  PROC DrawPart142()
    MoveL Offs(pOrigin,284.64,277.94,6.00),vTravel,z5,tPen\WObj:=wPaper;
    MoveL Offs(pOrigin,284.64,277.94,0.00),v60,z0,tPen\WObj:=wPaper;
    MoveL Offs(pOrigin,280.81,277.94,0.00),v40,fine,tPen\WObj:=wPaper;
    MoveL Offs(pOrigin,280.81,277.94,6.00),v60,z5,tPen\WObj:=wPaper;
    MoveL Offs(pOrigin,279.25,279.53,6.00),vTravel,z5,tPen\WObj:=wPaper;
    MoveL Offs(pOrigin,279.25,279.53,0.00),v60,z0,tPen\WObj:=wPaper;
    MoveL Offs(pOrigin,292.32,266.46,0.00),v40,z0,tPen\WObj:=wPaper;
    MoveL Offs(pOrigin,292.92,267.36,0.00),v40,z0,tPen\WObj:=wPaper;
    MoveL Offs(pOrigin,278.80,281.48,0.00),v40,z0,tPen\WObj:=wPaper;
    MoveL Offs(pOrigin,279.75,281.54,0.00),v40,z0,tPen\WObj:=wPaper;
    MoveL Offs(pOrigin,297.48,299.27,0.00),v40,z0,tPen\WObj:=wPaper;
    MoveL Offs(pOrigin,296.96,299.06,0.00),v40,z0,tPen\WObj:=wPaper;
    MoveL Offs(pOrigin,291.23,299.06,0.00),v40,z0,tPen\WObj:=wPaper;
    MoveL Offs(pOrigin,291.23,298.04,0.00),v40,z0,tPen\WObj:=wPaper;
    MoveL Offs(pOrigin,293.99,297.61,0.00),v40,z0,tPen\WObj:=wPaper;
    MoveL Offs(pOrigin,293.99,297.61,0.00),v40,z0,tPen\WObj:=wPaper;
    MoveL Offs(pOrigin,293.56,296.83,0.00),v40,z0,tPen\WObj:=wPaper;
    MoveL Offs(pOrigin,292.08,296.76,0.00),v40,z0,tPen\WObj:=wPaper;
    MoveL Offs(pOrigin,291.23,297.61,0.00),v40,fine,tPen\WObj:=wPaper;
    MoveL Offs(pOrigin,291.23,297.61,6.00),v60,z5,tPen\WObj:=wPaper;
    MoveL Offs(pOrigin,292.92,298.01,6.00),vTravel,z5,tPen\WObj:=wPaper;
    MoveL Offs(pOrigin,292.92,298.01,0.00),v60,z0,tPen\WObj:=wPaper;
    MoveL Offs(pOrigin,296.96,298.01,0.00),v40,z0,tPen\WObj:=wPaper;
    MoveL Offs(pOrigin,297.48,297.77,0.00),v40,z0,tPen\WObj:=wPaper;
    MoveL Offs(pOrigin,279.90,280.19,0.00),v40,fine,tPen\WObj:=wPaper;
    MoveL Offs(pOrigin,279.90,280.19,6.00),v60,z5,tPen\WObj:=wPaper;
    MoveL Offs(pOrigin,281.97,281.89,6.00),vTravel,z5,tPen\WObj:=wPaper;
    MoveL Offs(pOrigin,281.97,281.89,0.00),v60,z0,tPen\WObj:=wPaper;
    MoveL Offs(pOrigin,281.97,275.72,0.00),v40,z0,tPen\WObj:=wPaper;
    MoveL Offs(pOrigin,281.66,275.83,0.00),v40,z0,tPen\WObj:=wPaper;
    MoveL Offs(pOrigin,299.51,275.83,0.00),v40,z0,tPen\WObj:=wPaper;
    MoveL Offs(pOrigin,299.96,276.36,0.00),v40,z0,tPen\WObj:=wPaper;
    MoveL Offs(pOrigin,297.40,273.80,0.00),v40,z0,tPen\WObj:=wPaper;
    MoveL Offs(pOrigin,297.81,274.66,0.00),v40,z0,tPen\WObj:=wPaper;
    MoveL Offs(pOrigin,297.81,280.19,0.00),v40,z0,tPen\WObj:=wPaper;
    MoveL Offs(pOrigin,298.45,280.06,0.00),v40,z0,tPen\WObj:=wPaper;
    MoveL Offs(pOrigin,285.06,280.06,0.00),v40,z0,tPen\WObj:=wPaper;
    MoveL Offs(pOrigin,285.27,279.76,0.00),v40,z0,tPen\WObj:=wPaper;
    MoveL Offs(pOrigin,284.85,280.19,0.00),v40,z0,tPen\WObj:=wPaper;
    MoveL Offs(pOrigin,285.27,279.76,0.00),v40,z0,tPen\WObj:=wPaper;
    MoveL Offs(pOrigin,285.13,280.61,0.00),v40,z0,tPen\WObj:=wPaper;
    MoveL Offs(pOrigin,285.13,282.10,0.00),v40,z0,tPen\WObj:=wPaper;
    MoveL Offs(pOrigin,285.06,283.22,0.00),v40,z0,tPen\WObj:=wPaper;
    MoveL Offs(pOrigin,280.60,283.22,0.00),v40,z0,tPen\WObj:=wPaper;
    MoveL Offs(pOrigin,280.60,284.28,0.00),v40,z0,tPen\WObj:=wPaper;
    MoveL Offs(pOrigin,284.85,284.28,0.00),v40,z0,tPen\WObj:=wPaper;
    MoveL Offs(pOrigin,284.85,284.65,0.00),v40,z0,tPen\WObj:=wPaper;
    MoveL Offs(pOrigin,283.72,286.99,0.00),v40,z0,tPen\WObj:=wPaper;
    MoveL Offs(pOrigin,285.70,287.20,0.00),v40,z0,tPen\WObj:=wPaper;
    MoveL Offs(pOrigin,285.27,287.45,0.00),v40,z0,tPen\WObj:=wPaper;
    MoveL Offs(pOrigin,280.81,287.45,0.00),v40,z0,tPen\WObj:=wPaper;
    MoveL Offs(pOrigin,280.60,288.50,0.00),v40,z0,tPen\WObj:=wPaper;
    MoveL Offs(pOrigin,284.21,288.50,0.00),v40,z0,tPen\WObj:=wPaper;
    MoveL Offs(pOrigin,284.85,288.26,0.00),v40,z0,tPen\WObj:=wPaper;
    MoveL Offs(pOrigin,284.42,288.69,0.00),v40,z0,tPen\WObj:=wPaper;
    MoveL Offs(pOrigin,284.85,288.26,0.00),v40,fine,tPen\WObj:=wPaper;
    MoveL Offs(pOrigin,284.85,288.26,6.00),v60,z5,tPen\WObj:=wPaper;
    MoveL Offs(pOrigin,285.13,286.99,6.00),vTravel,z5,tPen\WObj:=wPaper;
    MoveL Offs(pOrigin,285.13,286.99,0.00),v60,z0,tPen\WObj:=wPaper;
    MoveL Offs(pOrigin,285.13,285.92,0.00),v40,z0,tPen\WObj:=wPaper;
    MoveL Offs(pOrigin,286.19,285.50,0.00),v40,z0,tPen\WObj:=wPaper;
    MoveL Offs(pOrigin,286.19,286.56,0.00),v40,fine,tPen\WObj:=wPaper;
    MoveL Offs(pOrigin,286.19,286.56,6.00),v60,z5,tPen\WObj:=wPaper;
    MoveL Offs(pOrigin,287.61,286.39,6.00),vTravel,z5,tPen\WObj:=wPaper;
    MoveL Offs(pOrigin,287.61,286.39,0.00),v60,z0,tPen\WObj:=wPaper;
    MoveL Offs(pOrigin,281.02,286.39,0.00),v40,z0,tPen\WObj:=wPaper;
    MoveL Offs(pOrigin,280.81,285.34,0.00),v40,z0,tPen\WObj:=wPaper;
    MoveL Offs(pOrigin,289.10,285.34,0.00),v40,z0,tPen\WObj:=wPaper;
    MoveL Offs(pOrigin,288.67,286.14,0.00),v40,z0,tPen\WObj:=wPaper;
    MoveL Offs(pOrigin,289.10,286.56,0.00),v40,z0,tPen\WObj:=wPaper;
    MoveL Offs(pOrigin,289.74,286.56,0.00),v40,z0,tPen\WObj:=wPaper;
    MoveL Offs(pOrigin,289.95,286.99,0.00),v40,z0,tPen\WObj:=wPaper;
    MoveL Offs(pOrigin,289.95,286.99,0.00),v40,z0,tPen\WObj:=wPaper;
    MoveL Offs(pOrigin,286.98,288.48,0.00),v40,z0,tPen\WObj:=wPaper;
    MoveL Offs(pOrigin,287.40,288.50,0.00),v40,z0,tPen\WObj:=wPaper;
    MoveL Offs(pOrigin,289.95,288.50,0.00),v40,z0,tPen\WObj:=wPaper;
    MoveL Offs(pOrigin,290.16,289.11,0.00),v40,z0,tPen\WObj:=wPaper;
    MoveL Offs(pOrigin,293.99,289.96,0.00),v40,z0,tPen\WObj:=wPaper;
    MoveL Offs(pOrigin,294.20,289.56,0.00),v40,z0,tPen\WObj:=wPaper;
    MoveL Offs(pOrigin,298.02,289.56,0.00),v40,fine,tPen\WObj:=wPaper;
    MoveL Offs(pOrigin,298.02,289.56,6.00),v60,z5,tPen\WObj:=wPaper;
    MoveL Offs(pOrigin,299.00,288.16,6.00),vTravel,z5,tPen\WObj:=wPaper;
    MoveL Offs(pOrigin,299.00,288.16,0.00),v60,z0,tPen\WObj:=wPaper;
    MoveL Offs(pOrigin,261.88,325.27,0.00),v40,z0,tPen\WObj:=wPaper;
    MoveL Offs(pOrigin,261.14,324.53,0.00),v40,z0,tPen\WObj:=wPaper;
    MoveL Offs(pOrigin,299.00,286.66,0.00),v40,z0,tPen\WObj:=wPaper;
    MoveL Offs(pOrigin,298.49,286.84,0.00),v40,z0,tPen\WObj:=wPaper;
    MoveL Offs(pOrigin,282.26,270.61,0.00),v40,z0,tPen\WObj:=wPaper;
    MoveL Offs(pOrigin,282.51,271.26,0.00),v40,z0,tPen\WObj:=wPaper;
    MoveL Offs(pOrigin,284.00,269.49,0.00),v40,z0,tPen\WObj:=wPaper;
    MoveL Offs(pOrigin,285.70,269.99,0.00),v40,z0,tPen\WObj:=wPaper;
    MoveL Offs(pOrigin,286.55,269.14,0.00),v40,z0,tPen\WObj:=wPaper;
    MoveL Offs(pOrigin,286.98,266.38,0.00),v40,z0,tPen\WObj:=wPaper;
    MoveL Offs(pOrigin,286.76,265.31,0.00),v40,z0,tPen\WObj:=wPaper;
    MoveL Offs(pOrigin,287.40,264.25,0.00),v40,fine,tPen\WObj:=wPaper;
    MoveL Offs(pOrigin,287.40,264.25,6.00),v60,z5,tPen\WObj:=wPaper;
    MoveL Offs(pOrigin,291.29,263.02,6.00),vTravel,z5,tPen\WObj:=wPaper;
    MoveL Offs(pOrigin,291.29,263.02,0.00),v60,z0,tPen\WObj:=wPaper;
    MoveL Offs(pOrigin,280.32,273.99,0.00),v40,z0,tPen\WObj:=wPaper;
    MoveL Offs(pOrigin,280.76,275.03,0.00),v40,z0,tPen\WObj:=wPaper;
    MoveL Offs(pOrigin,291.58,264.21,0.00),v40,fine,tPen\WObj:=wPaper;
    MoveL Offs(pOrigin,291.58,264.21,6.00),v60,z5,tPen\WObj:=wPaper;
    MoveL Offs(pOrigin,290.92,261.35,6.00),vTravel,z5,tPen\WObj:=wPaper;
    MoveL Offs(pOrigin,290.92,261.35,0.00),v60,z0,tPen\WObj:=wPaper;
    MoveL Offs(pOrigin,288.37,258.79,0.00),v40,fine,tPen\WObj:=wPaper;
    MoveL Offs(pOrigin,288.37,258.79,6.00),v60,z5,tPen\WObj:=wPaper;
    MoveL Offs(pOrigin,290.02,258.95,6.00),vTravel,z5,tPen\WObj:=wPaper;
    MoveL Offs(pOrigin,290.02,258.95,0.00),v60,z0,tPen\WObj:=wPaper;
    MoveL Offs(pOrigin,291.37,260.30,0.00),v40,z0,tPen\WObj:=wPaper;
    MoveL Offs(pOrigin,292.34,260.47,0.00),v40,z0,tPen\WObj:=wPaper;
    MoveL Offs(pOrigin,278.82,273.99,0.00),v40,fine,tPen\WObj:=wPaper;
    MoveL Offs(pOrigin,278.82,273.99,6.00),v60,z5,tPen\WObj:=wPaper;
    MoveL Offs(pOrigin,277.47,273.85,6.00),vTravel,z5,tPen\WObj:=wPaper;
    MoveL Offs(pOrigin,277.47,273.85,0.00),v60,z0,tPen\WObj:=wPaper;
    MoveL Offs(pOrigin,281.53,269.79,0.00),v40,fine,tPen\WObj:=wPaper;
    MoveL Offs(pOrigin,281.53,269.79,6.00),v60,z5,tPen\WObj:=wPaper;
    MoveL Offs(pOrigin,280.33,269.49,6.00),vTravel,z5,tPen\WObj:=wPaper;
    MoveL Offs(pOrigin,280.33,269.49,0.00),v60,z0,tPen\WObj:=wPaper;
    MoveL Offs(pOrigin,275.97,273.85,0.00),v40,z0,tPen\WObj:=wPaper;
    MoveL Offs(pOrigin,275.92,272.96,0.00),v40,z0,tPen\WObj:=wPaper;
  ENDPROC

  PROC DrawPart143()
    MoveL Offs(pOrigin,274.44,273.39,0.00),v40,fine,tPen\WObj:=wPaper;
    MoveL Offs(pOrigin,274.44,273.39,6.00),v60,z5,tPen\WObj:=wPaper;
    MoveL Offs(pOrigin,273.42,274.91,6.00),vTravel,z5,tPen\WObj:=wPaper;
    MoveL Offs(pOrigin,273.42,274.91,0.00),v60,z0,tPen\WObj:=wPaper;
    MoveL Offs(pOrigin,279.13,269.20,0.00),v40,z0,tPen\WObj:=wPaper;
    MoveL Offs(pOrigin,278.09,268.75,0.00),v40,z0,tPen\WObj:=wPaper;
    MoveL Offs(pOrigin,271.48,275.36,0.00),v40,fine,tPen\WObj:=wPaper;
    MoveL Offs(pOrigin,271.48,275.36,6.00),v60,z5,tPen\WObj:=wPaper;
    MoveL Offs(pOrigin,269.98,275.37,6.00),vTravel,z5,tPen\WObj:=wPaper;
    MoveL Offs(pOrigin,269.98,275.37,0.00),v60,z0,tPen\WObj:=wPaper;
    MoveL Offs(pOrigin,271.93,273.41,0.00),v40,z0,tPen\WObj:=wPaper;
    MoveL Offs(pOrigin,271.48,272.37,0.00),v40,z0,tPen\WObj:=wPaper;
    MoveL Offs(pOrigin,268.03,275.82,0.00),v40,z0,tPen\WObj:=wPaper;
    MoveL Offs(pOrigin,267.30,275.06,0.00),v40,z0,tPen\WObj:=wPaper;
    MoveL Offs(pOrigin,264.89,272.65,0.00),v40,z0,tPen\WObj:=wPaper;
    MoveL Offs(pOrigin,265.51,272.75,0.00),v40,z0,tPen\WObj:=wPaper;
    MoveL Offs(pOrigin,266.58,272.96,0.00),v40,z0,tPen\WObj:=wPaper;
    MoveL Offs(pOrigin,267.00,272.54,0.00),v40,z0,tPen\WObj:=wPaper;
    MoveL Offs(pOrigin,267.00,272.54,0.00),v40,z0,tPen\WObj:=wPaper;
    MoveL Offs(pOrigin,266.79,272.11,0.00),v40,z0,tPen\WObj:=wPaper;
    MoveL Offs(pOrigin,265.73,272.11,0.00),v40,z0,tPen\WObj:=wPaper;
    MoveL Offs(pOrigin,265.51,272.75,0.00),v40,z0,tPen\WObj:=wPaper;
    MoveL Offs(pOrigin,265.51,272.75,0.00),v40,z0,tPen\WObj:=wPaper;
    MoveL Offs(pOrigin,264.02,272.96,0.00),v40,z0,tPen\WObj:=wPaper;
    MoveL Offs(pOrigin,258.92,271.69,0.00),v40,z0,tPen\WObj:=wPaper;
    MoveL Offs(pOrigin,256.38,271.48,0.00),v40,z0,tPen\WObj:=wPaper;
    MoveL Offs(pOrigin,254.68,270.98,0.00),v40,z0,tPen\WObj:=wPaper;
    MoveL Offs(pOrigin,254.18,270.41,0.00),v40,z0,tPen\WObj:=wPaper;
    MoveL Offs(pOrigin,254.68,269.99,0.00),v40,z0,tPen\WObj:=wPaper;
    MoveL Offs(pOrigin,255.95,269.99,0.00),v40,z0,tPen\WObj:=wPaper;
    MoveL Offs(pOrigin,255.95,269.99,0.00),v40,z0,tPen\WObj:=wPaper;
    MoveL Offs(pOrigin,256.16,270.20,0.00),v40,z0,tPen\WObj:=wPaper;
    MoveL Offs(pOrigin,257.01,269.99,0.00),v40,z0,tPen\WObj:=wPaper;
    MoveL Offs(pOrigin,256.65,270.38,0.00),v40,z0,tPen\WObj:=wPaper;
    MoveL Offs(pOrigin,250.34,264.07,0.00),v40,fine,tPen\WObj:=wPaper;
    MoveL Offs(pOrigin,250.34,264.07,6.00),v60,z5,tPen\WObj:=wPaper;
    MoveL Offs(pOrigin,251.53,263.77,6.00),vTravel,z5,tPen\WObj:=wPaper;
    MoveL Offs(pOrigin,251.53,263.77,0.00),v60,z0,tPen\WObj:=wPaper;
    MoveL Offs(pOrigin,257.84,270.08,0.00),v40,z0,tPen\WObj:=wPaper;
    MoveL Offs(pOrigin,257.40,271.13,0.00),v40,z0,tPen\WObj:=wPaper;
    MoveL Offs(pOrigin,262.81,276.54,0.00),v40,z0,tPen\WObj:=wPaper;
    MoveL Offs(pOrigin,262.48,276.89,0.00),v40,z0,tPen\WObj:=wPaper;
    MoveL Offs(pOrigin,268.49,270.88,0.00),v40,z0,tPen\WObj:=wPaper;
    MoveL Offs(pOrigin,268.70,271.05,0.00),v40,z0,tPen\WObj:=wPaper;
    MoveL Offs(pOrigin,269.69,271.33,0.00),v40,z0,tPen\WObj:=wPaper;
    MoveL Offs(pOrigin,270.40,270.84,0.00),v40,z0,tPen\WObj:=wPaper;
    MoveL Offs(pOrigin,270.75,271.05,0.00),v40,z0,tPen\WObj:=wPaper;
    MoveL Offs(pOrigin,270.83,271.69,0.00),v40,z0,tPen\WObj:=wPaper;
    MoveL Offs(pOrigin,271.49,270.87,0.00),v40,z0,tPen\WObj:=wPaper;
    MoveL Offs(pOrigin,266.08,276.28,0.00),v40,z0,tPen\WObj:=wPaper;
    MoveL Offs(pOrigin,265.35,276.10,0.00),v40,z0,tPen\WObj:=wPaper;
    MoveL Offs(pOrigin,261.90,272.64,0.00),v40,z0,tPen\WObj:=wPaper;
    MoveL Offs(pOrigin,261.90,271.50,0.00),v40,z0,tPen\WObj:=wPaper;
    MoveL Offs(pOrigin,257.54,275.85,0.00),v40,z0,tPen\WObj:=wPaper;
    MoveL Offs(pOrigin,257.41,275.63,0.00),v40,z0,tPen\WObj:=wPaper;
    MoveL Offs(pOrigin,252.45,270.67,0.00),v40,fine,tPen\WObj:=wPaper;
    MoveL Offs(pOrigin,252.45,270.67,6.00),v60,z5,tPen\WObj:=wPaper;
    MoveL Offs(pOrigin,249.46,270.66,6.00),vTravel,z5,tPen\WObj:=wPaper;
    MoveL Offs(pOrigin,249.46,270.66,0.00),v60,z0,tPen\WObj:=wPaper;
    MoveL Offs(pOrigin,253.96,275.17,0.00),v40,z0,tPen\WObj:=wPaper;
    MoveL Offs(pOrigin,253.50,275.42,0.00),v40,z0,tPen\WObj:=wPaper;
    MoveL Offs(pOrigin,264.62,264.30,0.00),v40,z0,tPen\WObj:=wPaper;
    MoveL Offs(pOrigin,263.81,265.10,0.00),v40,z0,tPen\WObj:=wPaper;
    MoveL Offs(pOrigin,264.02,265.52,0.00),v40,z0,tPen\WObj:=wPaper;
    MoveL Offs(pOrigin,265.09,265.95,0.00),v40,z0,tPen\WObj:=wPaper;
    MoveL Offs(pOrigin,265.30,265.95,0.00),v40,z0,tPen\WObj:=wPaper;
    MoveL Offs(pOrigin,266.58,265.74,0.00),v40,z0,tPen\WObj:=wPaper;
    MoveL Offs(pOrigin,266.58,265.74,0.00),v40,z0,tPen\WObj:=wPaper;
    MoveL Offs(pOrigin,266.15,265.10,0.00),v40,z0,tPen\WObj:=wPaper;
    MoveL Offs(pOrigin,265.73,265.10,0.00),v40,z0,tPen\WObj:=wPaper;
    MoveL Offs(pOrigin,265.30,265.95,0.00),v40,z0,tPen\WObj:=wPaper;
    MoveL Offs(pOrigin,265.30,265.95,0.00),v40,z0,tPen\WObj:=wPaper;
    MoveL Offs(pOrigin,264.66,267.15,0.00),v40,z0,tPen\WObj:=wPaper;
    MoveL Offs(pOrigin,263.39,267.58,0.00),v40,z0,tPen\WObj:=wPaper;
    MoveL Offs(pOrigin,262.54,265.10,0.00),v40,z0,tPen\WObj:=wPaper;
    MoveL Offs(pOrigin,262.54,265.10,0.00),v40,z0,tPen\WObj:=wPaper;
    MoveL Offs(pOrigin,261.48,264.46,0.00),v40,z0,tPen\WObj:=wPaper;
    MoveL Offs(pOrigin,260.84,264.46,0.00),v40,z0,tPen\WObj:=wPaper;
    MoveL Offs(pOrigin,260.41,264.89,0.00),v40,z0,tPen\WObj:=wPaper;
    MoveL Offs(pOrigin,260.41,264.89,0.00),v40,z0,tPen\WObj:=wPaper;
    MoveL Offs(pOrigin,259.56,264.25,0.00),v40,z0,tPen\WObj:=wPaper;
    MoveL Offs(pOrigin,258.29,264.25,0.00),v40,z0,tPen\WObj:=wPaper;
    MoveL Offs(pOrigin,257.65,264.67,0.00),v40,z0,tPen\WObj:=wPaper;
    MoveL Offs(pOrigin,257.65,264.67,0.00),v40,z0,tPen\WObj:=wPaper;
    MoveL Offs(pOrigin,256.73,266.94,0.00),v40,z0,tPen\WObj:=wPaper;
    MoveL Offs(pOrigin,256.16,267.01,0.00),v40,z0,tPen\WObj:=wPaper;
    MoveL Offs(pOrigin,254.46,265.95,0.00),v40,z0,tPen\WObj:=wPaper;
    MoveL Offs(pOrigin,254.04,264.46,0.00),v40,z0,tPen\WObj:=wPaper;
    MoveL Offs(pOrigin,254.04,264.46,0.00),v40,z0,tPen\WObj:=wPaper;
    MoveL Offs(pOrigin,257.65,264.67,0.00),v40,z0,tPen\WObj:=wPaper;
    MoveL Offs(pOrigin,258.13,264.39,0.00),v40,z0,tPen\WObj:=wPaper;
    MoveL Offs(pOrigin,263.54,269.80,0.00),v40,z0,tPen\WObj:=wPaper;
    MoveL Offs(pOrigin,263.10,270.29,0.00),v40,z0,tPen\WObj:=wPaper;
    MoveL Offs(pOrigin,268.66,264.73,0.00),v40,z0,tPen\WObj:=wPaper;
    MoveL Offs(pOrigin,268.47,265.77,0.00),v40,z0,tPen\WObj:=wPaper;
    MoveL Offs(pOrigin,269.82,267.13,0.00),v40,z0,tPen\WObj:=wPaper;
    MoveL Offs(pOrigin,270.60,267.28,0.00),v40,z0,tPen\WObj:=wPaper;
    MoveL Offs(pOrigin,272.55,265.32,0.00),v40,z0,tPen\WObj:=wPaper;
    MoveL Offs(pOrigin,271.66,264.73,0.00),v40,z0,tPen\WObj:=wPaper;
    MoveL Offs(pOrigin,267.15,269.23,0.00),v40,z0,tPen\WObj:=wPaper;
    MoveL Offs(pOrigin,266.98,268.76,0.00),v40,z0,tPen\WObj:=wPaper;
    MoveL Offs(pOrigin,264.27,266.06,0.00),v40,z0,tPen\WObj:=wPaper;
    MoveL Offs(pOrigin,265.30,266.33,0.00),v40,z0,tPen\WObj:=wPaper;
    MoveL Offs(pOrigin,268.91,266.33,0.00),v40,z0,tPen\WObj:=wPaper;
    MoveL Offs(pOrigin,269.55,266.16,0.00),v40,z0,tPen\WObj:=wPaper;
    MoveL Offs(pOrigin,268.70,265.74,0.00),v40,z0,tPen\WObj:=wPaper;
    MoveL Offs(pOrigin,266.58,265.74,0.00),v40,z0,tPen\WObj:=wPaper;
    MoveL Offs(pOrigin,266.67,265.47,0.00),v40,z0,tPen\WObj:=wPaper;
    MoveL Offs(pOrigin,268.92,267.72,0.00),v40,z0,tPen\WObj:=wPaper;
    MoveL Offs(pOrigin,268.49,267.38,0.00),v40,z0,tPen\WObj:=wPaper;
    MoveL Offs(pOrigin,255.95,267.38,0.00),v40,z0,tPen\WObj:=wPaper;
    MoveL Offs(pOrigin,255.74,266.48,0.00),v40,z0,tPen\WObj:=wPaper;
    MoveL Offs(pOrigin,259.34,270.09,0.00),v40,z0,tPen\WObj:=wPaper;
    MoveL Offs(pOrigin,259.14,269.77,0.00),v40,z0,tPen\WObj:=wPaper;
    MoveL Offs(pOrigin,262.75,269.56,0.00),v40,z0,tPen\WObj:=wPaper;
    MoveL Offs(pOrigin,267.64,268.36,0.00),v40,z0,tPen\WObj:=wPaper;
    MoveL Offs(pOrigin,269.98,266.16,0.00),v40,z0,tPen\WObj:=wPaper;
    MoveL Offs(pOrigin,271.25,266.23,0.00),v40,z0,tPen\WObj:=wPaper;
    MoveL Offs(pOrigin,272.95,267.65,0.00),v40,fine,tPen\WObj:=wPaper;
    MoveL Offs(pOrigin,272.95,267.65,6.00),v60,z5,tPen\WObj:=wPaper;
  ENDPROC

  PROC DrawPart144()
    MoveL Offs(pOrigin,274.01,266.38,6.00),vTravel,z5,tPen\WObj:=wPaper;
    MoveL Offs(pOrigin,274.01,266.38,0.00),v60,z0,tPen\WObj:=wPaper;
    MoveL Offs(pOrigin,272.52,265.95,0.00),v40,z0,tPen\WObj:=wPaper;
    MoveL Offs(pOrigin,271.46,266.16,0.00),v40,z0,tPen\WObj:=wPaper;
    MoveL Offs(pOrigin,270.57,266.38,0.00),v40,z0,tPen\WObj:=wPaper;
    MoveL Offs(pOrigin,269.66,265.48,0.00),v40,z0,tPen\WObj:=wPaper;
    MoveL Offs(pOrigin,270.31,264.58,0.00),v40,z0,tPen\WObj:=wPaper;
    MoveL Offs(pOrigin,265.05,269.84,0.00),v40,z0,tPen\WObj:=wPaper;
    MoveL Offs(pOrigin,264.73,269.51,0.00),v40,z0,tPen\WObj:=wPaper;
    MoveL Offs(pOrigin,259.32,264.10,0.00),v40,z0,tPen\WObj:=wPaper;
    MoveL Offs(pOrigin,259.68,263.26,0.00),v40,z0,tPen\WObj:=wPaper;
    MoveL Offs(pOrigin,247.96,274.98,0.00),v40,fine,tPen\WObj:=wPaper;
    MoveL Offs(pOrigin,247.96,274.98,6.00),v60,z5,tPen\WObj:=wPaper;
    MoveL Offs(pOrigin,249.46,274.98,6.00),vTravel,z5,tPen\WObj:=wPaper;
    MoveL Offs(pOrigin,249.46,274.98,0.00),v60,z0,tPen\WObj:=wPaper;
    MoveL Offs(pOrigin,260.88,263.56,0.00),v40,z0,tPen\WObj:=wPaper;
    MoveL Offs(pOrigin,261.12,264.40,0.00),v40,z0,tPen\WObj:=wPaper;
    MoveL Offs(pOrigin,265.78,269.06,0.00),v40,z0,tPen\WObj:=wPaper;
    MoveL Offs(pOrigin,264.88,268.44,0.00),v40,z0,tPen\WObj:=wPaper;
    MoveL Offs(pOrigin,257.23,268.44,0.00),v40,z0,tPen\WObj:=wPaper;
    MoveL Offs(pOrigin,257.68,267.86,0.00),v40,z0,tPen\WObj:=wPaper;
    MoveL Offs(pOrigin,257.68,266.59,0.00),v40,z0,tPen\WObj:=wPaper;
    MoveL Offs(pOrigin,257.23,266.33,0.00),v40,z0,tPen\WObj:=wPaper;
    MoveL Offs(pOrigin,262.75,266.33,0.00),v40,z0,tPen\WObj:=wPaper;
    MoveL Offs(pOrigin,262.54,265.74,0.00),v40,z0,tPen\WObj:=wPaper;
    MoveL Offs(pOrigin,261.48,266.16,0.00),v40,z0,tPen\WObj:=wPaper;
    MoveL Offs(pOrigin,260.84,265.52,0.00),v40,z0,tPen\WObj:=wPaper;
    MoveL Offs(pOrigin,260.41,265.52,0.00),v40,z0,tPen\WObj:=wPaper;
    MoveL Offs(pOrigin,260.41,265.52,0.00),v40,z0,tPen\WObj:=wPaper;
    MoveL Offs(pOrigin,258.92,265.60,0.00),v40,z0,tPen\WObj:=wPaper;
    MoveL Offs(pOrigin,258.15,266.38,0.00),v40,z0,tPen\WObj:=wPaper;
    MoveL Offs(pOrigin,258.36,267.58,0.00),v40,z0,tPen\WObj:=wPaper;
    MoveL Offs(pOrigin,259.14,267.86,0.00),v40,z0,tPen\WObj:=wPaper;
    MoveL Offs(pOrigin,258.73,267.86,0.00),v40,z0,tPen\WObj:=wPaper;
    MoveL Offs(pOrigin,258.73,265.31,0.00),v40,z0,tPen\WObj:=wPaper;
    MoveL Offs(pOrigin,257.86,265.27,0.00),v40,z0,tPen\WObj:=wPaper;
    MoveL Offs(pOrigin,262.11,265.27,0.00),v40,z0,tPen\WObj:=wPaper;
    MoveL Offs(pOrigin,262.33,264.67,0.00),v40,z0,tPen\WObj:=wPaper;
    MoveL Offs(pOrigin,262.75,265.10,0.00),v40,z0,tPen\WObj:=wPaper;
    MoveL Offs(pOrigin,263.81,265.10,0.00),v40,z0,tPen\WObj:=wPaper;
    MoveL Offs(pOrigin,263.81,265.10,0.00),v40,z0,tPen\WObj:=wPaper;
    MoveL Offs(pOrigin,264.02,264.46,0.00),v40,z0,tPen\WObj:=wPaper;
    MoveL Offs(pOrigin,264.88,264.46,0.00),v40,z0,tPen\WObj:=wPaper;
    MoveL Offs(pOrigin,265.51,265.10,0.00),v40,z0,tPen\WObj:=wPaper;
    MoveL Offs(pOrigin,265.67,264.74,0.00),v40,z0,tPen\WObj:=wPaper;
    MoveL Offs(pOrigin,254.70,275.71,0.00),v40,fine,tPen\WObj:=wPaper;
    MoveL Offs(pOrigin,254.70,275.71,6.00),v60,z5,tPen\WObj:=wPaper;
    MoveL Offs(pOrigin,256.04,275.86,6.00),vTravel,z5,tPen\WObj:=wPaper;
    MoveL Offs(pOrigin,256.04,275.86,0.00),v60,z0,tPen\WObj:=wPaper;
    MoveL Offs(pOrigin,267.01,264.89,0.00),v40,fine,tPen\WObj:=wPaper;
    MoveL Offs(pOrigin,267.01,264.89,6.00),v60,z5,tPen\WObj:=wPaper;
    MoveL Offs(pOrigin,266.13,266.59,6.00),vTravel,z5,tPen\WObj:=wPaper;
    MoveL Offs(pOrigin,266.13,266.59,0.00),v60,z0,tPen\WObj:=wPaper;
    MoveL Offs(pOrigin,266.13,267.65,0.00),v40,fine,tPen\WObj:=wPaper;
    MoveL Offs(pOrigin,266.13,267.65,6.00),v60,z5,tPen\WObj:=wPaper;
    MoveL Offs(pOrigin,264.24,267.44,6.00),vTravel,z5,tPen\WObj:=wPaper;
    MoveL Offs(pOrigin,264.24,267.44,0.00),v60,z0,tPen\WObj:=wPaper;
    MoveL Offs(pOrigin,264.66,267.01,0.00),v40,z0,tPen\WObj:=wPaper;
    MoveL Offs(pOrigin,264.24,267.44,0.00),v40,fine,tPen\WObj:=wPaper;
    MoveL Offs(pOrigin,264.24,267.44,6.00),v60,z5,tPen\WObj:=wPaper;
    MoveL Offs(pOrigin,265.17,265.46,6.00),vTravel,z5,tPen\WObj:=wPaper;
    MoveL Offs(pOrigin,265.17,265.46,0.00),v60,z0,tPen\WObj:=wPaper;
    MoveL Offs(pOrigin,268.02,268.32,0.00),v40,fine,tPen\WObj:=wPaper;
    MoveL Offs(pOrigin,268.02,268.32,6.00),v60,z5,tPen\WObj:=wPaper;
    MoveL Offs(pOrigin,270.44,270.42,6.00),vTravel,z5,tPen\WObj:=wPaper;
    MoveL Offs(pOrigin,270.44,270.42,0.00),v60,z0,tPen\WObj:=wPaper;
    MoveL Offs(pOrigin,263.98,276.88,0.00),v40,fine,tPen\WObj:=wPaper;
    MoveL Offs(pOrigin,263.98,276.88,6.00),v60,z5,tPen\WObj:=wPaper;
    MoveL Offs(pOrigin,262.33,276.36,6.00),vTravel,z5,tPen\WObj:=wPaper;
    MoveL Offs(pOrigin,262.33,276.36,0.00),v60,z0,tPen\WObj:=wPaper;
    MoveL Offs(pOrigin,262.11,275.73,0.00),v40,z0,tPen\WObj:=wPaper;
    MoveL Offs(pOrigin,261.05,275.94,0.00),v40,z0,tPen\WObj:=wPaper;
    MoveL Offs(pOrigin,261.05,275.94,0.00),v40,z0,tPen\WObj:=wPaper;
    MoveL Offs(pOrigin,261.48,276.58,0.00),v40,z0,tPen\WObj:=wPaper;
    MoveL Offs(pOrigin,262.33,276.36,0.00),v40,fine,tPen\WObj:=wPaper;
    MoveL Offs(pOrigin,262.33,276.36,6.00),v60,z5,tPen\WObj:=wPaper;
    MoveL Offs(pOrigin,261.13,276.74,6.00),vTravel,z5,tPen\WObj:=wPaper;
    MoveL Offs(pOrigin,261.13,276.74,0.00),v60,z0,tPen\WObj:=wPaper;
    MoveL Offs(pOrigin,266.39,271.48,0.00),v40,z0,tPen\WObj:=wPaper;
    MoveL Offs(pOrigin,267.00,272.11,0.00),v40,z0,tPen\WObj:=wPaper;
    MoveL Offs(pOrigin,267.42,271.69,0.00),v40,z0,tPen\WObj:=wPaper;
    MoveL Offs(pOrigin,268.27,271.69,0.00),v40,z0,tPen\WObj:=wPaper;
    MoveL Offs(pOrigin,268.27,272.11,0.00),v40,z0,tPen\WObj:=wPaper;
    MoveL Offs(pOrigin,268.27,272.11,0.00),v40,z0,tPen\WObj:=wPaper;
    MoveL Offs(pOrigin,268.06,272.54,0.00),v40,z0,tPen\WObj:=wPaper;
    MoveL Offs(pOrigin,267.00,272.54,0.00),v40,z0,tPen\WObj:=wPaper;
    MoveL Offs(pOrigin,266.39,272.66,0.00),v40,z0,tPen\WObj:=wPaper;
    MoveL Offs(pOrigin,268.34,274.61,0.00),v40,z0,tPen\WObj:=wPaper;
    MoveL Offs(pOrigin,268.49,274.45,0.00),v40,z0,tPen\WObj:=wPaper;
    MoveL Offs(pOrigin,268.06,273.81,0.00),v40,z0,tPen\WObj:=wPaper;
    MoveL Offs(pOrigin,267.00,273.81,0.00),v40,z0,tPen\WObj:=wPaper;
    MoveL Offs(pOrigin,266.58,274.45,0.00),v40,z0,tPen\WObj:=wPaper;
    MoveL Offs(pOrigin,266.79,274.66,0.00),v40,z0,tPen\WObj:=wPaper;
    MoveL Offs(pOrigin,268.06,274.66,0.00),v40,fine,tPen\WObj:=wPaper;
    MoveL Offs(pOrigin,268.06,274.66,6.00),v60,z5,tPen\WObj:=wPaper;
    MoveL Offs(pOrigin,269.24,274.01,6.00),vTravel,z5,tPen\WObj:=wPaper;
    MoveL Offs(pOrigin,269.24,274.01,0.00),v60,z0,tPen\WObj:=wPaper;
    MoveL Offs(pOrigin,267.74,272.51,0.00),v40,z0,tPen\WObj:=wPaper;
    MoveL Offs(pOrigin,268.27,272.11,0.00),v40,z0,tPen\WObj:=wPaper;
    MoveL Offs(pOrigin,269.55,271.62,0.00),v40,z0,tPen\WObj:=wPaper;
    MoveL Offs(pOrigin,270.75,272.11,0.00),v40,z0,tPen\WObj:=wPaper;
    MoveL Offs(pOrigin,269.76,274.24,0.00),v40,z0,tPen\WObj:=wPaper;
    MoveL Offs(pOrigin,269.84,273.12,0.00),v40,z0,tPen\WObj:=wPaper;
    MoveL Offs(pOrigin,268.79,272.07,0.00),v40,fine,tPen\WObj:=wPaper;
    MoveL Offs(pOrigin,268.79,272.07,6.00),v60,z5,tPen\WObj:=wPaper;
    MoveL Offs(pOrigin,265.73,273.72,6.00),vTravel,z5,tPen\WObj:=wPaper;
    MoveL Offs(pOrigin,265.73,273.72,0.00),v60,z0,tPen\WObj:=wPaper;
    MoveL Offs(pOrigin,264.66,273.72,0.00),v40,fine,tPen\WObj:=wPaper;
    MoveL Offs(pOrigin,264.66,273.72,6.00),v60,z5,tPen\WObj:=wPaper;
    MoveL Offs(pOrigin,264.60,271.79,6.00),vTravel,z5,tPen\WObj:=wPaper;
    MoveL Offs(pOrigin,264.60,271.79,0.00),v60,z0,tPen\WObj:=wPaper;
    MoveL Offs(pOrigin,260.09,276.30,0.00),v40,z0,tPen\WObj:=wPaper;
    MoveL Offs(pOrigin,261.01,276.24,0.00),v40,z0,tPen\WObj:=wPaper;
    MoveL Offs(pOrigin,245.83,261.06,0.00),v40,z0,tPen\WObj:=wPaper;
    MoveL Offs(pOrigin,246.28,260.01,0.00),v40,z0,tPen\WObj:=wPaper;
    MoveL Offs(pOrigin,249.28,263.02,0.00),v40,z0,tPen\WObj:=wPaper;
    MoveL Offs(pOrigin,248.51,263.83,0.00),v40,z0,tPen\WObj:=wPaper;
    MoveL Offs(pOrigin,247.88,263.19,0.00),v40,z0,tPen\WObj:=wPaper;
    MoveL Offs(pOrigin,247.88,263.19,0.00),v40,z0,tPen\WObj:=wPaper;
    MoveL Offs(pOrigin,247.02,263.61,0.00),v40,z0,tPen\WObj:=wPaper;
  ENDPROC

  PROC DrawPart145()
    MoveL Offs(pOrigin,246.81,264.46,0.00),v40,z0,tPen\WObj:=wPaper;
    MoveL Offs(pOrigin,246.81,264.46,0.00),v40,z0,tPen\WObj:=wPaper;
    MoveL Offs(pOrigin,246.81,265.95,0.00),v40,z0,tPen\WObj:=wPaper;
    MoveL Offs(pOrigin,246.60,265.95,0.00),v40,z0,tPen\WObj:=wPaper;
    MoveL Offs(pOrigin,246.30,266.00,0.00),v40,z0,tPen\WObj:=wPaper;
    MoveL Offs(pOrigin,244.79,264.50,0.00),v40,z0,tPen\WObj:=wPaper;
    MoveL Offs(pOrigin,245.32,264.89,0.00),v40,z0,tPen\WObj:=wPaper;
    MoveL Offs(pOrigin,245.75,265.10,0.00),v40,z0,tPen\WObj:=wPaper;
    MoveL Offs(pOrigin,245.75,265.95,0.00),v40,z0,tPen\WObj:=wPaper;
    MoveL Offs(pOrigin,245.55,266.75,0.00),v40,z0,tPen\WObj:=wPaper;
    MoveL Offs(pOrigin,244.35,265.55,0.00),v40,z0,tPen\WObj:=wPaper;
    MoveL Offs(pOrigin,244.69,266.16,0.00),v40,z0,tPen\WObj:=wPaper;
    MoveL Offs(pOrigin,243.41,266.38,0.00),v40,z0,tPen\WObj:=wPaper;
    MoveL Offs(pOrigin,240.23,266.16,0.00),v40,z0,tPen\WObj:=wPaper;
    MoveL Offs(pOrigin,238.10,265.31,0.00),v40,z0,tPen\WObj:=wPaper;
    MoveL Offs(pOrigin,237.25,263.83,0.00),v40,z0,tPen\WObj:=wPaper;
    MoveL Offs(pOrigin,237.25,263.83,0.00),v40,z0,tPen\WObj:=wPaper;
    MoveL Offs(pOrigin,235.98,264.67,0.00),v40,z0,tPen\WObj:=wPaper;
    MoveL Offs(pOrigin,235.34,265.52,0.00),v40,fine,tPen\WObj:=wPaper;
    MoveL Offs(pOrigin,235.34,265.52,6.00),v60,z5,tPen\WObj:=wPaper;
    MoveL Offs(pOrigin,235.98,264.22,6.00),vTravel,z5,tPen\WObj:=wPaper;
    MoveL Offs(pOrigin,235.98,264.22,0.00),v60,z0,tPen\WObj:=wPaper;
    MoveL Offs(pOrigin,222.16,264.22,0.00),v40,z0,tPen\WObj:=wPaper;
    MoveL Offs(pOrigin,221.13,264.73,0.00),v40,z0,tPen\WObj:=wPaper;
    MoveL Offs(pOrigin,215.27,258.87,0.00),v40,z0,tPen\WObj:=wPaper;
    MoveL Offs(pOrigin,215.36,259.15,0.00),v40,z0,tPen\WObj:=wPaper;
    MoveL Offs(pOrigin,214.73,257.45,0.00),v40,z0,tPen\WObj:=wPaper;
    MoveL Offs(pOrigin,213.66,256.60,0.00),v40,fine,tPen\WObj:=wPaper;
    MoveL Offs(pOrigin,213.66,256.60,6.00),v60,z5,tPen\WObj:=wPaper;
    MoveL Offs(pOrigin,214.46,257.71,6.00),vTravel,z5,tPen\WObj:=wPaper;
    MoveL Offs(pOrigin,214.46,257.71,0.00),v60,z0,tPen\WObj:=wPaper;
    MoveL Offs(pOrigin,212.95,259.21,0.00),v40,z0,tPen\WObj:=wPaper;
    MoveL Offs(pOrigin,212.60,260.21,0.00),v40,z0,tPen\WObj:=wPaper;
    MoveL Offs(pOrigin,213.88,259.79,0.00),v40,z0,tPen\WObj:=wPaper;
    MoveL Offs(pOrigin,214.51,259.15,0.00),v40,z0,tPen\WObj:=wPaper;
    MoveL Offs(pOrigin,214.51,259.15,0.00),v40,z0,tPen\WObj:=wPaper;
    MoveL Offs(pOrigin,213.66,258.51,0.00),v40,z0,tPen\WObj:=wPaper;
    MoveL Offs(pOrigin,211.75,258.51,0.00),v40,fine,tPen\WObj:=wPaper;
    MoveL Offs(pOrigin,211.75,258.51,6.00),v60,z5,tPen\WObj:=wPaper;
    MoveL Offs(pOrigin,212.18,260.21,6.00),vTravel,z5,tPen\WObj:=wPaper;
    MoveL Offs(pOrigin,212.18,260.21,0.00),v60,z0,tPen\WObj:=wPaper;
    MoveL Offs(pOrigin,213.10,261.70,0.00),v40,z0,tPen\WObj:=wPaper;
    MoveL Offs(pOrigin,213.24,262.98,0.00),v40,z0,tPen\WObj:=wPaper;
    MoveL Offs(pOrigin,213.24,262.98,0.00),v40,z0,tPen\WObj:=wPaper;
    MoveL Offs(pOrigin,213.88,263.68,0.00),v40,z0,tPen\WObj:=wPaper;
    MoveL Offs(pOrigin,214.73,263.90,0.00),v40,z0,tPen\WObj:=wPaper;
    MoveL Offs(pOrigin,215.15,264.67,0.00),v40,z0,tPen\WObj:=wPaper;
    MoveL Offs(pOrigin,217.49,266.09,0.00),v40,z0,tPen\WObj:=wPaper;
    MoveL Offs(pOrigin,221.52,267.23,0.00),v40,z0,tPen\WObj:=wPaper;
    MoveL Offs(pOrigin,221.52,267.23,0.00),v40,z0,tPen\WObj:=wPaper;
    MoveL Offs(pOrigin,221.74,266.80,0.00),v40,z0,tPen\WObj:=wPaper;
    MoveL Offs(pOrigin,222.80,267.01,0.00),v40,z0,tPen\WObj:=wPaper;
    MoveL Offs(pOrigin,221.73,266.83,0.00),v40,z0,tPen\WObj:=wPaper;
    MoveL Offs(pOrigin,226.84,271.94,0.00),v40,z0,tPen\WObj:=wPaper;
    MoveL Offs(pOrigin,226.69,272.35,0.00),v40,z0,tPen\WObj:=wPaper;
    MoveL Offs(pOrigin,239.02,260.03,0.00),v40,z0,tPen\WObj:=wPaper;
    MoveL Offs(pOrigin,238.19,259.39,0.00),v40,z0,tPen\WObj:=wPaper;
    MoveL Offs(pOrigin,235.48,256.68,0.00),v40,z0,tPen\WObj:=wPaper;
    MoveL Offs(pOrigin,236.19,256.39,0.00),v40,z0,tPen\WObj:=wPaper;
    MoveL Offs(pOrigin,236.19,257.24,0.00),v40,z0,tPen\WObj:=wPaper;
    MoveL Offs(pOrigin,236.82,257.88,0.00),v40,z0,tPen\WObj:=wPaper;
    MoveL Offs(pOrigin,236.82,257.88,0.00),v40,z0,tPen\WObj:=wPaper;
    MoveL Offs(pOrigin,237.68,257.02,0.00),v40,z0,tPen\WObj:=wPaper;
    MoveL Offs(pOrigin,237.60,256.17,0.00),v40,z0,tPen\WObj:=wPaper;
    MoveL Offs(pOrigin,237.04,255.75,0.00),v40,z0,tPen\WObj:=wPaper;
    MoveL Offs(pOrigin,237.04,255.75,0.00),v40,z0,tPen\WObj:=wPaper;
    MoveL Offs(pOrigin,236.19,256.39,0.00),v40,z0,tPen\WObj:=wPaper;
    MoveL Offs(pOrigin,236.19,256.39,0.00),v40,z0,tPen\WObj:=wPaper;
    MoveL Offs(pOrigin,235.69,255.96,0.00),v40,z0,tPen\WObj:=wPaper;
    MoveL Offs(pOrigin,235.62,255.11,0.00),v40,z0,tPen\WObj:=wPaper;
    MoveL Offs(pOrigin,236.40,255.18,0.00),v40,z0,tPen\WObj:=wPaper;
    MoveL Offs(pOrigin,237.04,255.75,0.00),v40,z0,tPen\WObj:=wPaper;
    MoveL Offs(pOrigin,237.83,255.24,0.00),v40,z0,tPen\WObj:=wPaper;
    MoveL Offs(pOrigin,221.45,271.62,0.00),v40,z0,tPen\WObj:=wPaper;
    MoveL Offs(pOrigin,221.75,271.32,0.00),v40,z0,tPen\WObj:=wPaper;
    MoveL Offs(pOrigin,213.63,263.21,0.00),v40,z0,tPen\WObj:=wPaper;
    MoveL Offs(pOrigin,213.24,263.40,0.00),v40,z0,tPen\WObj:=wPaper;
    MoveL Offs(pOrigin,213.10,264.89,0.00),v40,z0,tPen\WObj:=wPaper;
    MoveL Offs(pOrigin,214.51,266.59,0.00),v40,z0,tPen\WObj:=wPaper;
    MoveL Offs(pOrigin,219.19,267.86,0.00),v40,z0,tPen\WObj:=wPaper;
    MoveL Offs(pOrigin,219.19,267.86,0.00),v40,z0,tPen\WObj:=wPaper;
    MoveL Offs(pOrigin,220.89,268.08,0.00),v40,z0,tPen\WObj:=wPaper;
    MoveL Offs(pOrigin,221.74,267.86,0.00),v40,fine,tPen\WObj:=wPaper;
    MoveL Offs(pOrigin,221.74,267.86,6.00),v60,z5,tPen\WObj:=wPaper;
    MoveL Offs(pOrigin,222.38,268.92,6.00),vTravel,z5,tPen\WObj:=wPaper;
    MoveL Offs(pOrigin,222.38,268.92,0.00),v60,z0,tPen\WObj:=wPaper;
    MoveL Offs(pOrigin,225.56,269.14,0.00),v40,z0,tPen\WObj:=wPaper;
    MoveL Offs(pOrigin,225.56,269.14,0.00),v40,z0,tPen\WObj:=wPaper;
    MoveL Offs(pOrigin,228.96,269.35,0.00),v40,z0,tPen\WObj:=wPaper;
    MoveL Offs(pOrigin,229.81,268.71,0.00),v40,z0,tPen\WObj:=wPaper;
    MoveL Offs(pOrigin,230.45,268.71,0.00),v40,z0,tPen\WObj:=wPaper;
    MoveL Offs(pOrigin,231.09,268.08,0.00),v40,z0,tPen\WObj:=wPaper;
    MoveL Offs(pOrigin,232.15,268.08,0.00),v40,z0,tPen\WObj:=wPaper;
    MoveL Offs(pOrigin,232.79,268.50,0.00),v40,z0,tPen\WObj:=wPaper;
    MoveL Offs(pOrigin,232.79,269.14,0.00),v40,z0,tPen\WObj:=wPaper;
    MoveL Offs(pOrigin,231.73,269.56,0.00),v40,z0,tPen\WObj:=wPaper;
    MoveL Offs(pOrigin,231.09,269.50,0.00),v40,z0,tPen\WObj:=wPaper;
    MoveL Offs(pOrigin,216.64,269.50,0.00),v40,fine,tPen\WObj:=wPaper;
    MoveL Offs(pOrigin,216.64,269.50,6.00),v60,z5,tPen\WObj:=wPaper;
    MoveL Offs(pOrigin,216.00,268.44,6.00),vTravel,z5,tPen\WObj:=wPaper;
    MoveL Offs(pOrigin,216.00,268.44,0.00),v60,z0,tPen\WObj:=wPaper;
    MoveL Offs(pOrigin,220.46,268.44,0.00),v40,fine,tPen\WObj:=wPaper;
    MoveL Offs(pOrigin,220.46,268.44,6.00),v60,z5,tPen\WObj:=wPaper;
    MoveL Offs(pOrigin,219.40,267.38,6.00),vTravel,z5,tPen\WObj:=wPaper;
    MoveL Offs(pOrigin,219.40,267.38,0.00),v60,z0,tPen\WObj:=wPaper;
    MoveL Offs(pOrigin,216.64,267.38,0.00),v40,fine,tPen\WObj:=wPaper;
    MoveL Offs(pOrigin,216.64,267.38,6.00),v60,z5,tPen\WObj:=wPaper;
    MoveL Offs(pOrigin,215.79,265.31,6.00),vTravel,z5,tPen\WObj:=wPaper;
    MoveL Offs(pOrigin,215.79,265.31,0.00),v60,z0,tPen\WObj:=wPaper;
    MoveL Offs(pOrigin,216.21,265.52,0.00),v40,z0,tPen\WObj:=wPaper;
    MoveL Offs(pOrigin,215.79,265.31,0.00),v40,z0,tPen\WObj:=wPaper;
    MoveL Offs(pOrigin,216.53,264.60,0.00),v40,z0,tPen\WObj:=wPaper;
    MoveL Offs(pOrigin,212.78,268.35,0.00),v40,z0,tPen\WObj:=wPaper;
    MoveL Offs(pOrigin,213.82,268.80,0.00),v40,z0,tPen\WObj:=wPaper;
    MoveL Offs(pOrigin,217.58,265.04,0.00),v40,fine,tPen\WObj:=wPaper;
    MoveL Offs(pOrigin,217.58,265.04,6.00),v60,z5,tPen\WObj:=wPaper;
    MoveL Offs(pOrigin,218.78,265.34,6.00),vTravel,z5,tPen\WObj:=wPaper;
    MoveL Offs(pOrigin,218.78,265.34,0.00),v60,z0,tPen\WObj:=wPaper;
    MoveL Offs(pOrigin,214.57,269.54,0.00),v40,fine,tPen\WObj:=wPaper;
    MoveL Offs(pOrigin,214.57,269.54,6.00),v60,z5,tPen\WObj:=wPaper;
  ENDPROC

  PROC DrawPart146()
    MoveL Offs(pOrigin,211.58,268.06,6.00),vTravel,z5,tPen\WObj:=wPaper;
    MoveL Offs(pOrigin,211.58,268.06,0.00),v60,z0,tPen\WObj:=wPaper;
    MoveL Offs(pOrigin,215.48,264.15,0.00),v40,z0,tPen\WObj:=wPaper;
    MoveL Offs(pOrigin,214.89,263.25,0.00),v40,z0,tPen\WObj:=wPaper;
    MoveL Offs(pOrigin,210.53,267.61,0.00),v40,z0,tPen\WObj:=wPaper;
    MoveL Offs(pOrigin,209.48,267.16,0.00),v40,z0,tPen\WObj:=wPaper;
    MoveL Offs(pOrigin,210.84,265.81,0.00),v40,z0,tPen\WObj:=wPaper;
    MoveL Offs(pOrigin,209.94,265.21,0.00),v40,z0,tPen\WObj:=wPaper;
    MoveL Offs(pOrigin,208.44,266.72,0.00),v40,fine,tPen\WObj:=wPaper;
    MoveL Offs(pOrigin,208.44,266.72,6.00),v60,z5,tPen\WObj:=wPaper;
    MoveL Offs(pOrigin,206.75,266.78,6.00),vTravel,z5,tPen\WObj:=wPaper;
    MoveL Offs(pOrigin,206.75,266.78,0.00),v60,z0,tPen\WObj:=wPaper;
    MoveL Offs(pOrigin,201.79,261.82,0.00),v40,fine,tPen\WObj:=wPaper;
    MoveL Offs(pOrigin,201.79,261.82,6.00),v60,z5,tPen\WObj:=wPaper;
    MoveL Offs(pOrigin,202.77,262.55,6.00),vTravel,z5,tPen\WObj:=wPaper;
    MoveL Offs(pOrigin,202.77,262.55,0.00),v60,z0,tPen\WObj:=wPaper;
    MoveL Offs(pOrigin,202.77,268.08,0.00),v40,z0,tPen\WObj:=wPaper;
    MoveL Offs(pOrigin,201.71,268.29,0.00),v40,z0,tPen\WObj:=wPaper;
    MoveL Offs(pOrigin,201.71,269.35,0.00),v40,z0,tPen\WObj:=wPaper;
    MoveL Offs(pOrigin,200.65,268.92,0.00),v40,z0,tPen\WObj:=wPaper;
    MoveL Offs(pOrigin,200.65,263.82,0.00),v40,z0,tPen\WObj:=wPaper;
    MoveL Offs(pOrigin,200.00,263.02,0.00),v40,z0,tPen\WObj:=wPaper;
    MoveL Offs(pOrigin,206.31,269.33,0.00),v40,z0,tPen\WObj:=wPaper;
    MoveL Offs(pOrigin,205.80,269.50,0.00),v40,z0,tPen\WObj:=wPaper;
    MoveL Offs(pOrigin,197.73,269.50,0.00),v40,z0,tPen\WObj:=wPaper;
    MoveL Offs(pOrigin,197.17,269.15,0.00),v40,z0,tPen\WObj:=wPaper;
    MoveL Offs(pOrigin,204.84,276.81,0.00),v40,z0,tPen\WObj:=wPaper;
    MoveL Offs(pOrigin,205.56,277.06,0.00),v40,z0,tPen\WObj:=wPaper;
    MoveL Offs(pOrigin,189.78,292.84,0.00),v40,z0,tPen\WObj:=wPaper;
    MoveL Offs(pOrigin,190.36,293.70,0.00),v40,z0,tPen\WObj:=wPaper;
    MoveL Offs(pOrigin,196.37,299.71,0.00),v40,z0,tPen\WObj:=wPaper;
    MoveL Offs(pOrigin,195.60,300.16,0.00),v40,z0,tPen\WObj:=wPaper;
    MoveL Offs(pOrigin,196.02,300.80,0.00),v40,z0,tPen\WObj:=wPaper;
    MoveL Offs(pOrigin,195.60,300.16,0.00),v40,z0,tPen\WObj:=wPaper;
    MoveL Offs(pOrigin,195.18,299.52,0.00),v40,z0,tPen\WObj:=wPaper;
    MoveL Offs(pOrigin,195.39,299.95,0.00),v40,z0,tPen\WObj:=wPaper;
    MoveL Offs(pOrigin,195.18,299.52,0.00),v40,fine,tPen\WObj:=wPaper;
    MoveL Offs(pOrigin,195.18,299.52,6.00),v60,z5,tPen\WObj:=wPaper;
    MoveL Offs(pOrigin,193.69,300.12,6.00),vTravel,z5,tPen\WObj:=wPaper;
    MoveL Offs(pOrigin,193.69,300.12,0.00),v60,z0,tPen\WObj:=wPaper;
    MoveL Offs(pOrigin,191.56,300.12,0.00),v40,z0,tPen\WObj:=wPaper;
    MoveL Offs(pOrigin,192.21,300.80,0.00),v40,z0,tPen\WObj:=wPaper;
    MoveL Offs(pOrigin,192.21,296.97,0.00),v40,z0,tPen\WObj:=wPaper;
    MoveL Offs(pOrigin,192.20,295.90,0.00),v40,z0,tPen\WObj:=wPaper;
    MoveL Offs(pOrigin,194.54,295.90,0.00),v40,z0,tPen\WObj:=wPaper;
    MoveL Offs(pOrigin,195.46,295.81,0.00),v40,z0,tPen\WObj:=wPaper;
    MoveL Offs(pOrigin,190.95,291.30,0.00),v40,z0,tPen\WObj:=wPaper;
    MoveL Offs(pOrigin,190.93,291.66,0.00),v40,z0,tPen\WObj:=wPaper;
    MoveL Offs(pOrigin,191.35,290.60,0.00),v40,z0,tPen\WObj:=wPaper;
    MoveL Offs(pOrigin,190.50,286.56,0.00),v40,z0,tPen\WObj:=wPaper;
    MoveL Offs(pOrigin,190.93,282.74,0.00),v40,z0,tPen\WObj:=wPaper;
    MoveL Offs(pOrigin,193.12,276.36,0.00),v40,z0,tPen\WObj:=wPaper;
    MoveL Offs(pOrigin,197.58,269.14,0.00),v40,z0,tPen\WObj:=wPaper;
    MoveL Offs(pOrigin,197.87,267.86,0.00),v40,z0,tPen\WObj:=wPaper;
    MoveL Offs(pOrigin,198.79,266.38,0.00),v40,z0,tPen\WObj:=wPaper;
    MoveL Offs(pOrigin,198.72,264.53,0.00),v40,z0,tPen\WObj:=wPaper;
    MoveL Offs(pOrigin,196.45,262.76,0.00),v40,z0,tPen\WObj:=wPaper;
    MoveL Offs(pOrigin,195.18,260.21,0.00),v40,z0,tPen\WObj:=wPaper;
    MoveL Offs(pOrigin,194.75,257.24,0.00),v40,z0,tPen\WObj:=wPaper;
    MoveL Offs(pOrigin,194.96,253.62,0.00),v40,z0,tPen\WObj:=wPaper;
    MoveL Offs(pOrigin,196.17,250.23,0.00),v40,z0,tPen\WObj:=wPaper;
    MoveL Offs(pOrigin,199.78,244.27,0.00),v40,z0,tPen\WObj:=wPaper;
    MoveL Offs(pOrigin,200.91,240.45,0.00),v40,z0,tPen\WObj:=wPaper;
    MoveL Offs(pOrigin,200.27,240.02,0.00),v40,z0,tPen\WObj:=wPaper;
    MoveL Offs(pOrigin,184.98,237.26,0.00),v40,z0,tPen\WObj:=wPaper;
    MoveL Offs(pOrigin,178.18,235.35,0.00),v40,z0,tPen\WObj:=wPaper;
    MoveL Offs(pOrigin,172.65,233.08,0.00),v40,z0,tPen\WObj:=wPaper;
    MoveL Offs(pOrigin,169.04,230.89,0.00),v40,z0,tPen\WObj:=wPaper;
    MoveL Offs(pOrigin,166.91,229.19,0.00),v40,z0,tPen\WObj:=wPaper;
    MoveL Offs(pOrigin,164.79,226.85,0.00),v40,z0,tPen\WObj:=wPaper;
    MoveL Offs(pOrigin,163.23,224.51,0.00),v40,z0,tPen\WObj:=wPaper;
    MoveL Offs(pOrigin,161.74,221.54,0.00),v40,z0,tPen\WObj:=wPaper;
    MoveL Offs(pOrigin,160.54,217.50,0.00),v40,z0,tPen\WObj:=wPaper;
    MoveL Offs(pOrigin,159.90,212.61,0.00),v40,z0,tPen\WObj:=wPaper;
    MoveL Offs(pOrigin,159.48,205.18,0.00),v40,z0,tPen\WObj:=wPaper;
    MoveL Offs(pOrigin,159.40,193.27,0.00),v40,z0,tPen\WObj:=wPaper;
    MoveL Offs(pOrigin,143.75,188.46,0.00),v40,z0,tPen\WObj:=wPaper;
    MoveL Offs(pOrigin,141.41,187.11,0.00),v40,z0,tPen\WObj:=wPaper;
    MoveL Offs(pOrigin,138.93,183.93,0.00),v40,z0,tPen\WObj:=wPaper;
    MoveL Offs(pOrigin,137.38,179.68,0.00),v40,z0,tPen\WObj:=wPaper;
    MoveL Offs(pOrigin,136.10,173.09,0.00),v40,z0,tPen\WObj:=wPaper;
    MoveL Offs(pOrigin,133.12,166.07,0.00),v40,z0,tPen\WObj:=wPaper;
    MoveL Offs(pOrigin,132.63,160.76,0.00),v40,z0,tPen\WObj:=wPaper;
    MoveL Offs(pOrigin,130.57,158.85,0.00),v40,z0,tPen\WObj:=wPaper;
    MoveL Offs(pOrigin,129.51,156.73,0.00),v40,z0,tPen\WObj:=wPaper;
    MoveL Offs(pOrigin,129.37,151.20,0.00),v40,z0,tPen\WObj:=wPaper;
    MoveL Offs(pOrigin,127.39,148.86,0.00),v40,z0,tPen\WObj:=wPaper;
    MoveL Offs(pOrigin,126.32,146.95,0.00),v40,z0,tPen\WObj:=wPaper;
    MoveL Offs(pOrigin,126.11,140.57,0.00),v40,z0,tPen\WObj:=wPaper;
    MoveL Offs(pOrigin,125.76,139.51,0.00),v40,z0,tPen\WObj:=wPaper;
    MoveL Offs(pOrigin,123.49,136.54,0.00),v40,z0,tPen\WObj:=wPaper;
    MoveL Offs(pOrigin,123.00,133.99,0.00),v40,z0,tPen\WObj:=wPaper;
    MoveL Offs(pOrigin,120.80,133.28,0.00),v40,z0,tPen\WObj:=wPaper;
    MoveL Offs(pOrigin,118.39,131.01,0.00),v40,z0,tPen\WObj:=wPaper;
    MoveL Offs(pOrigin,117.40,128.25,0.00),v40,z0,tPen\WObj:=wPaper;
    MoveL Offs(pOrigin,116.55,122.51,0.00),v40,z0,tPen\WObj:=wPaper;
    MoveL Offs(pOrigin,115.56,119.11,0.00),v40,z0,tPen\WObj:=wPaper;
    MoveL Offs(pOrigin,113.79,116.35,0.00),v40,z0,tPen\WObj:=wPaper;
    MoveL Offs(pOrigin,109.75,111.68,0.00),v40,z0,tPen\WObj:=wPaper;
    MoveL Offs(pOrigin,107.77,108.70,0.00),v40,z0,tPen\WObj:=wPaper;
    MoveL Offs(pOrigin,105.43,103.18,0.00),v40,z0,tPen\WObj:=wPaper;
    MoveL Offs(pOrigin,102.60,94.25,0.00),v40,z0,tPen\WObj:=wPaper;
    MoveL Offs(pOrigin,99.76,91.70,0.00),v40,z0,tPen\WObj:=wPaper;
    MoveL Offs(pOrigin,98.20,89.57,0.00),v40,z0,tPen\WObj:=wPaper;
    MoveL Offs(pOrigin,94.52,81.29,0.00),v40,z0,tPen\WObj:=wPaper;
    MoveL Offs(pOrigin,90.98,75.55,0.00),v40,z0,tPen\WObj:=wPaper;
    MoveL Offs(pOrigin,89.56,71.51,0.00),v40,z0,tPen\WObj:=wPaper;
    MoveL Offs(pOrigin,89.14,68.75,0.00),v40,z0,tPen\WObj:=wPaper;
    MoveL Offs(pOrigin,89.35,64.07,0.00),v40,z0,tPen\WObj:=wPaper;
    MoveL Offs(pOrigin,90.62,58.34,0.00),v40,z0,tPen\WObj:=wPaper;
    MoveL Offs(pOrigin,92.32,53.88,0.00),v40,z0,tPen\WObj:=wPaper;
    MoveL Offs(pOrigin,92.54,48.14,0.00),v40,z0,tPen\WObj:=wPaper;
    MoveL Offs(pOrigin,92.89,46.86,0.00),v40,z0,tPen\WObj:=wPaper;
    MoveL Offs(pOrigin,94.24,44.53,0.00),v40,z0,tPen\WObj:=wPaper;
    MoveL Offs(pOrigin,97.07,41.83,0.00),v40,z0,tPen\WObj:=wPaper;
    MoveL Offs(pOrigin,96.79,41.97,0.00),v40,z0,tPen\WObj:=wPaper;
    MoveL Offs(pOrigin,96.36,42.46,0.00),v40,z0,tPen\WObj:=wPaper;
    MoveL Offs(pOrigin,98.49,42.46,0.00),v40,z0,tPen\WObj:=wPaper;
    MoveL Offs(pOrigin,98.91,42.61,0.00),v40,z0,tPen\WObj:=wPaper;
    MoveL Offs(pOrigin,99.97,41.90,0.00),v40,z0,tPen\WObj:=wPaper;
  ENDPROC

  PROC DrawPart147()
    MoveL Offs(pOrigin,102.74,40.91,0.00),v40,z0,tPen\WObj:=wPaper;
    MoveL Offs(pOrigin,105.50,40.28,0.00),v40,z0,tPen\WObj:=wPaper;
    MoveL Offs(pOrigin,106.70,40.35,0.00),v40,z0,tPen\WObj:=wPaper;
    MoveL Offs(pOrigin,106.63,41.34,0.00),v40,z0,tPen\WObj:=wPaper;
    MoveL Offs(pOrigin,105.43,43.46,0.00),v40,z0,tPen\WObj:=wPaper;
    MoveL Offs(pOrigin,104.86,45.59,0.00),v40,z0,tPen\WObj:=wPaper;
    MoveL Offs(pOrigin,104.86,49.84,0.00),v40,z0,tPen\WObj:=wPaper;
    MoveL Offs(pOrigin,105.29,50.47,0.00),v40,z0,tPen\WObj:=wPaper;
    MoveL Offs(pOrigin,105.29,50.47,0.00),v40,z0,tPen\WObj:=wPaper;
    MoveL Offs(pOrigin,106.70,54.94,0.00),v40,z0,tPen\WObj:=wPaper;
    MoveL Offs(pOrigin,107.84,56.85,0.00),v40,fine,tPen\WObj:=wPaper;
    MoveL Offs(pOrigin,107.84,56.85,6.00),v60,z5,tPen\WObj:=wPaper;
    MoveL Offs(pOrigin,106.32,55.21,6.00),vTravel,z5,tPen\WObj:=wPaper;
    MoveL Offs(pOrigin,106.32,55.21,0.00),v60,z0,tPen\WObj:=wPaper;
    MoveL Offs(pOrigin,107.22,54.31,0.00),v40,fine,tPen\WObj:=wPaper;
    MoveL Offs(pOrigin,107.22,54.31,6.00),v60,z5,tPen\WObj:=wPaper;
    MoveL Offs(pOrigin,106.93,53.12,6.00),vTravel,z5,tPen\WObj:=wPaper;
    MoveL Offs(pOrigin,106.93,53.12,0.00),v60,z0,tPen\WObj:=wPaper;
    MoveL Offs(pOrigin,105.73,54.32,0.00),v40,z0,tPen\WObj:=wPaper;
    MoveL Offs(pOrigin,105.28,53.27,0.00),v40,z0,tPen\WObj:=wPaper;
    MoveL Offs(pOrigin,106.63,51.92,0.00),v40,fine,tPen\WObj:=wPaper;
    MoveL Offs(pOrigin,106.63,51.92,6.00),v60,z5,tPen\WObj:=wPaper;
    MoveL Offs(pOrigin,106.49,50.57,6.00),vTravel,z5,tPen\WObj:=wPaper;
    MoveL Offs(pOrigin,106.49,50.57,0.00),v60,z0,tPen\WObj:=wPaper;
    MoveL Offs(pOrigin,104.83,52.22,0.00),v40,z0,tPen\WObj:=wPaper;
    MoveL Offs(pOrigin,104.39,51.18,0.00),v40,z0,tPen\WObj:=wPaper;
    MoveL Offs(pOrigin,106.34,49.22,0.00),v40,z0,tPen\WObj:=wPaper;
    MoveL Offs(pOrigin,105.72,49.26,0.00),v40,z0,tPen\WObj:=wPaper;
    MoveL Offs(pOrigin,104.52,48.06,0.00),v40,z0,tPen\WObj:=wPaper;
    MoveL Offs(pOrigin,103.95,48.63,0.00),v40,z0,tPen\WObj:=wPaper;
    MoveL Offs(pOrigin,106.80,45.78,0.00),v40,z0,tPen\WObj:=wPaper;
    MoveL Offs(pOrigin,106.31,45.37,0.00),v40,z0,tPen\WObj:=wPaper;
    MoveL Offs(pOrigin,104.95,44.02,0.00),v40,z0,tPen\WObj:=wPaper;
    MoveL Offs(pOrigin,104.41,43.69,0.00),v40,z0,tPen\WObj:=wPaper;
    MoveL Offs(pOrigin,113.28,34.82,0.00),v40,fine,tPen\WObj:=wPaper;
    MoveL Offs(pOrigin,113.28,34.82,6.00),v60,z5,tPen\WObj:=wPaper;
    MoveL Offs(pOrigin,111.93,34.67,6.00),vTravel,z5,tPen\WObj:=wPaper;
    MoveL Offs(pOrigin,111.93,34.67,0.00),v60,z0,tPen\WObj:=wPaper;
    MoveL Offs(pOrigin,104.87,41.74,0.00),v40,z0,tPen\WObj:=wPaper;
    MoveL Offs(pOrigin,105.85,41.92,0.00),v40,z0,tPen\WObj:=wPaper;
    MoveL Offs(pOrigin,107.20,43.28,0.00),v40,z0,tPen\WObj:=wPaper;
    MoveL Offs(pOrigin,106.99,43.04,0.00),v40,z0,tPen\WObj:=wPaper;
    MoveL Offs(pOrigin,106.78,43.46,0.00),v40,z0,tPen\WObj:=wPaper;
    MoveL Offs(pOrigin,106.99,43.04,0.00),v40,z0,tPen\WObj:=wPaper;
    MoveL Offs(pOrigin,107.20,42.46,0.00),v40,z0,tPen\WObj:=wPaper;
    MoveL Offs(pOrigin,106.14,42.46,0.00),v40,z0,tPen\WObj:=wPaper;
    MoveL Offs(pOrigin,105.93,42.19,0.00),v40,z0,tPen\WObj:=wPaper;
    MoveL Offs(pOrigin,105.71,42.61,0.00),v40,z0,tPen\WObj:=wPaper;
    MoveL Offs(pOrigin,105.93,42.19,0.00),v40,z0,tPen\WObj:=wPaper;
    MoveL Offs(pOrigin,105.40,42.97,0.00),v40,z0,tPen\WObj:=wPaper;
    MoveL Offs(pOrigin,106.75,44.32,0.00),v40,fine,tPen\WObj:=wPaper;
    MoveL Offs(pOrigin,106.75,44.32,6.00),v60,z5,tPen\WObj:=wPaper;
    MoveL Offs(pOrigin,107.71,43.38,6.00),vTravel,z5,tPen\WObj:=wPaper;
    MoveL Offs(pOrigin,107.71,43.38,0.00),v60,z0,tPen\WObj:=wPaper;
    MoveL Offs(pOrigin,103.80,47.28,0.00),v40,z0,tPen\WObj:=wPaper;
    MoveL Offs(pOrigin,104.51,46.56,0.00),v40,z0,tPen\WObj:=wPaper;
    MoveL Offs(pOrigin,105.87,47.92,0.00),v40,z0,tPen\WObj:=wPaper;
    MoveL Offs(pOrigin,106.65,47.42,0.00),v40,z0,tPen\WObj:=wPaper;
    MoveL Offs(pOrigin,104.24,49.83,0.00),v40,z0,tPen\WObj:=wPaper;
    MoveL Offs(pOrigin,104.82,49.86,0.00),v40,z0,tPen\WObj:=wPaper;
    MoveL Offs(pOrigin,105.72,50.76,0.00),v40,z0,tPen\WObj:=wPaper;
    MoveL Offs(pOrigin,105.29,50.47,0.00),v40,z0,tPen\WObj:=wPaper;
    MoveL Offs(pOrigin,105.71,50.05,0.00),v40,z0,tPen\WObj:=wPaper;
    MoveL Offs(pOrigin,105.71,47.08,0.00),v40,z0,tPen\WObj:=wPaper;
    MoveL Offs(pOrigin,106.28,44.74,0.00),v40,z0,tPen\WObj:=wPaper;
    MoveL Offs(pOrigin,107.62,42.40,0.00),v40,z0,tPen\WObj:=wPaper;
    MoveL Offs(pOrigin,108.97,40.98,0.00),v40,z0,tPen\WObj:=wPaper;
    MoveL Offs(pOrigin,107.41,42.40,0.00),v40,z0,tPen\WObj:=wPaper;
    MoveL Offs(pOrigin,107.80,42.38,0.00),v40,z0,tPen\WObj:=wPaper;
    MoveL Offs(pOrigin,100.58,35.17,0.00),v40,fine,tPen\WObj:=wPaper;
    MoveL Offs(pOrigin,100.58,35.17,6.00),v60,z5,tPen\WObj:=wPaper;
    MoveL Offs(pOrigin,102.53,35.62,6.00),vTravel,z5,tPen\WObj:=wPaper;
    MoveL Offs(pOrigin,102.53,35.62,0.00),v60,z0,tPen\WObj:=wPaper;
    MoveL Offs(pOrigin,108.54,41.63,0.00),v40,z0,tPen\WObj:=wPaper;
    MoveL Offs(pOrigin,109.21,41.87,0.00),v40,z0,tPen\WObj:=wPaper;
    MoveL Offs(pOrigin,115.97,35.11,0.00),v40,z0,tPen\WObj:=wPaper;
    MoveL Offs(pOrigin,116.34,36.24,0.00),v40,z0,tPen\WObj:=wPaper;
    MoveL Offs(pOrigin,116.55,35.81,0.00),v40,z0,tPen\WObj:=wPaper;
    MoveL Offs(pOrigin,117.19,35.81,0.00),v40,z0,tPen\WObj:=wPaper;
    MoveL Offs(pOrigin,117.61,36.45,0.00),v40,z0,tPen\WObj:=wPaper;
    MoveL Offs(pOrigin,117.61,36.45,0.00),v40,z0,tPen\WObj:=wPaper;
    MoveL Offs(pOrigin,117.61,36.24,0.00),v40,z0,tPen\WObj:=wPaper;
    MoveL Offs(pOrigin,119.74,36.66,0.00),v40,z0,tPen\WObj:=wPaper;
    MoveL Offs(pOrigin,119.74,36.66,0.00),v40,z0,tPen\WObj:=wPaper;
    MoveL Offs(pOrigin,120.38,37.09,0.00),v40,z0,tPen\WObj:=wPaper;
    MoveL Offs(pOrigin,121.37,36.88,0.00),v40,z0,tPen\WObj:=wPaper;
    MoveL Offs(pOrigin,120.80,36.24,0.00),v40,z0,tPen\WObj:=wPaper;
    MoveL Offs(pOrigin,119.95,36.31,0.00),v40,z0,tPen\WObj:=wPaper;
    MoveL Offs(pOrigin,119.74,36.66,0.00),v40,z0,tPen\WObj:=wPaper;
    MoveL Offs(pOrigin,120.02,35.55,0.00),v40,z0,tPen\WObj:=wPaper;
    MoveL Offs(pOrigin,110.40,45.17,0.00),v40,z0,tPen\WObj:=wPaper;
    MoveL Offs(pOrigin,111.30,45.76,0.00),v40,z0,tPen\WObj:=wPaper;
    MoveL Offs(pOrigin,121.36,35.69,0.00),v40,fine,tPen\WObj:=wPaper;
    MoveL Offs(pOrigin,121.36,35.69,6.00),v60,z5,tPen\WObj:=wPaper;
    MoveL Offs(pOrigin,122.56,35.99,6.00),vTravel,z5,tPen\WObj:=wPaper;
    MoveL Offs(pOrigin,122.56,35.99,0.00),v60,z0,tPen\WObj:=wPaper;
    MoveL Offs(pOrigin,112.79,45.76,0.00),v40,z0,tPen\WObj:=wPaper;
    MoveL Offs(pOrigin,113.50,45.09,0.00),v40,z0,tPen\WObj:=wPaper;
    MoveL Offs(pOrigin,110.64,42.24,0.00),v40,z0,tPen\WObj:=wPaper;
    MoveL Offs(pOrigin,109.96,42.62,0.00),v40,z0,tPen\WObj:=wPaper;
    MoveL Offs(pOrigin,117.17,35.41,0.00),v40,fine,tPen\WObj:=wPaper;
    MoveL Offs(pOrigin,117.17,35.41,6.00),v60,z5,tPen\WObj:=wPaper;
    MoveL Offs(pOrigin,116.62,37.76,6.00),vTravel,z5,tPen\WObj:=wPaper;
    MoveL Offs(pOrigin,116.62,37.76,0.00),v60,z0,tPen\WObj:=wPaper;
    MoveL Offs(pOrigin,122.48,43.62,0.00),v40,z0,tPen\WObj:=wPaper;
    MoveL Offs(pOrigin,122.08,43.51,0.00),v40,z0,tPen\WObj:=wPaper;
    MoveL Offs(pOrigin,119.95,43.51,0.00),v40,z0,tPen\WObj:=wPaper;
    MoveL Offs(pOrigin,119.33,43.46,0.00),v40,z0,tPen\WObj:=wPaper;
    MoveL Offs(pOrigin,121.59,45.72,0.00),v40,z0,tPen\WObj:=wPaper;
    MoveL Offs(pOrigin,121.22,45.62,0.00),v40,z0,tPen\WObj:=wPaper;
    MoveL Offs(pOrigin,119.74,45.62,0.00),v40,z0,tPen\WObj:=wPaper;
    MoveL Offs(pOrigin,119.19,44.81,0.00),v40,z0,tPen\WObj:=wPaper;
    MoveL Offs(pOrigin,121.44,47.06,0.00),v40,z0,tPen\WObj:=wPaper;
    MoveL Offs(pOrigin,121.78,47.23,0.00),v40,z0,tPen\WObj:=wPaper;
    MoveL Offs(pOrigin,118.62,50.38,0.00),v40,z0,tPen\WObj:=wPaper;
    MoveL Offs(pOrigin,119.21,50.80,0.00),v40,z0,tPen\WObj:=wPaper;
    MoveL Offs(pOrigin,126.72,58.32,0.00),v40,z0,tPen\WObj:=wPaper;
    MoveL Offs(pOrigin,126.11,58.34,0.00),v40,z0,tPen\WObj:=wPaper;
    MoveL Offs(pOrigin,124.62,57.70,0.00),v40,z0,tPen\WObj:=wPaper;
    MoveL Offs(pOrigin,122.22,54.30,0.00),v40,z0,tPen\WObj:=wPaper;
  ENDPROC

  PROC DrawPart148()
    MoveL Offs(pOrigin,122.07,52.17,0.00),v40,z0,tPen\WObj:=wPaper;
    MoveL Offs(pOrigin,121.01,48.56,0.00),v40,z0,tPen\WObj:=wPaper;
    MoveL Offs(pOrigin,121.22,46.22,0.00),v40,z0,tPen\WObj:=wPaper;
    MoveL Offs(pOrigin,122.64,43.04,0.00),v40,z0,tPen\WObj:=wPaper;
    MoveL Offs(pOrigin,124.62,40.70,0.00),v40,z0,tPen\WObj:=wPaper;
    MoveL Offs(pOrigin,125.90,40.28,0.00),v40,z0,tPen\WObj:=wPaper;
    MoveL Offs(pOrigin,126.32,40.91,0.00),v40,z0,tPen\WObj:=wPaper;
    MoveL Offs(pOrigin,124.70,43.46,0.00),v40,z0,tPen\WObj:=wPaper;
    MoveL Offs(pOrigin,123.78,47.50,0.00),v40,z0,tPen\WObj:=wPaper;
    MoveL Offs(pOrigin,123.99,51.54,0.00),v40,z0,tPen\WObj:=wPaper;
    MoveL Offs(pOrigin,124.55,53.88,0.00),v40,z0,tPen\WObj:=wPaper;
    MoveL Offs(pOrigin,125.05,54.09,0.00),v40,z0,tPen\WObj:=wPaper;
    MoveL Offs(pOrigin,125.21,53.82,0.00),v40,z0,tPen\WObj:=wPaper;
    MoveL Offs(pOrigin,123.85,52.46,0.00),v40,fine,tPen\WObj:=wPaper;
    MoveL Offs(pOrigin,123.85,52.46,6.00),v60,z5,tPen\WObj:=wPaper;
    MoveL Offs(pOrigin,125.05,52.17,6.00),vTravel,z5,tPen\WObj:=wPaper;
    MoveL Offs(pOrigin,125.05,52.17,0.00),v60,z0,tPen\WObj:=wPaper;
    MoveL Offs(pOrigin,123.70,50.82,0.00),v40,fine,tPen\WObj:=wPaper;
    MoveL Offs(pOrigin,123.70,50.82,6.00),v60,z5,tPen\WObj:=wPaper;
    MoveL Offs(pOrigin,125.05,50.67,6.00),vTravel,z5,tPen\WObj:=wPaper;
    MoveL Offs(pOrigin,125.05,50.67,0.00),v60,z0,tPen\WObj:=wPaper;
    MoveL Offs(pOrigin,123.40,49.02,0.00),v40,fine,tPen\WObj:=wPaper;
    MoveL Offs(pOrigin,123.40,49.02,6.00),v60,z5,tPen\WObj:=wPaper;
    MoveL Offs(pOrigin,123.69,47.82,6.00),vTravel,z5,tPen\WObj:=wPaper;
    MoveL Offs(pOrigin,123.69,47.82,0.00),v60,z0,tPen\WObj:=wPaper;
    MoveL Offs(pOrigin,125.19,49.32,0.00),v40,z0,tPen\WObj:=wPaper;
    MoveL Offs(pOrigin,125.82,49.16,0.00),v40,z0,tPen\WObj:=wPaper;
    MoveL Offs(pOrigin,119.35,55.62,0.00),v40,z0,tPen\WObj:=wPaper;
    MoveL Offs(pOrigin,119.82,55.90,0.00),v40,z0,tPen\WObj:=wPaper;
    MoveL Offs(pOrigin,132.59,68.67,0.00),v40,z0,tPen\WObj:=wPaper;
    MoveL Offs(pOrigin,132.64,69.21,0.00),v40,z0,tPen\WObj:=wPaper;
    MoveL Offs(pOrigin,135.20,66.66,0.00),v40,z0,tPen\WObj:=wPaper;
    MoveL Offs(pOrigin,134.45,65.91,0.00),v40,z0,tPen\WObj:=wPaper;
    MoveL Offs(pOrigin,131.75,68.62,0.00),v40,z0,tPen\WObj:=wPaper;
    MoveL Offs(pOrigin,132.28,67.80,0.00),v40,z0,tPen\WObj:=wPaper;
    MoveL Offs(pOrigin,135.68,67.80,0.00),v40,fine,tPen\WObj:=wPaper;
    MoveL Offs(pOrigin,135.68,67.80,6.00),v60,z5,tPen\WObj:=wPaper;
    MoveL Offs(pOrigin,133.98,66.74,6.00),vTravel,z5,tPen\WObj:=wPaper;
    MoveL Offs(pOrigin,133.98,66.74,0.00),v60,z0,tPen\WObj:=wPaper;
    MoveL Offs(pOrigin,130.36,66.74,0.00),v40,z0,tPen\WObj:=wPaper;
    MoveL Offs(pOrigin,130.96,66.84,0.00),v40,z0,tPen\WObj:=wPaper;
    MoveL Offs(pOrigin,130.96,65.14,0.00),v40,z0,tPen\WObj:=wPaper;
    MoveL Offs(pOrigin,131.21,64.63,0.00),v40,z0,tPen\WObj:=wPaper;
    MoveL Offs(pOrigin,126.96,64.63,0.00),v40,z0,tPen\WObj:=wPaper;
    MoveL Offs(pOrigin,126.22,65.19,0.00),v40,z0,tPen\WObj:=wPaper;
    MoveL Offs(pOrigin,129.82,61.58,0.00),v40,z0,tPen\WObj:=wPaper;
    MoveL Offs(pOrigin,129.51,62.38,0.00),v40,z0,tPen\WObj:=wPaper;
    MoveL Offs(pOrigin,129.94,62.80,0.00),v40,z0,tPen\WObj:=wPaper;
    MoveL Offs(pOrigin,129.51,62.38,0.00),v40,z0,tPen\WObj:=wPaper;
    MoveL Offs(pOrigin,130.42,62.48,0.00),v40,z0,tPen\WObj:=wPaper;
    MoveL Offs(pOrigin,126.96,65.94,0.00),v40,z0,tPen\WObj:=wPaper;
    MoveL Offs(pOrigin,127.86,66.53,0.00),v40,z0,tPen\WObj:=wPaper;
    MoveL Offs(pOrigin,131.17,63.23,0.00),v40,z0,tPen\WObj:=wPaper;
    MoveL Offs(pOrigin,131.91,63.97,0.00),v40,z0,tPen\WObj:=wPaper;
    MoveL Offs(pOrigin,128.91,66.98,0.00),v40,z0,tPen\WObj:=wPaper;
    MoveL Offs(pOrigin,129.59,67.16,0.00),v40,z0,tPen\WObj:=wPaper;
    MoveL Offs(pOrigin,120.73,58.30,0.00),v40,z0,tPen\WObj:=wPaper;
    MoveL Offs(pOrigin,121.22,58.30,0.00),v40,z0,tPen\WObj:=wPaper;
    MoveL Offs(pOrigin,122.71,58.30,0.00),v40,z0,tPen\WObj:=wPaper;
    MoveL Offs(pOrigin,123.27,57.86,0.00),v40,z0,tPen\WObj:=wPaper;
    MoveL Offs(pOrigin,119.67,54.25,0.00),v40,z0,tPen\WObj:=wPaper;
    MoveL Offs(pOrigin,119.21,54.28,0.00),v40,z0,tPen\WObj:=wPaper;
    MoveL Offs(pOrigin,127.17,46.31,0.00),v40,z0,tPen\WObj:=wPaper;
    MoveL Offs(pOrigin,126.23,45.88,0.00),v40,z0,tPen\WObj:=wPaper;
    MoveL Offs(pOrigin,124.28,43.93,0.00),v40,z0,tPen\WObj:=wPaper;
    MoveL Offs(pOrigin,124.41,44.57,0.00),v40,z0,tPen\WObj:=wPaper;
    MoveL Offs(pOrigin,126.32,44.57,0.00),v40,z0,tPen\WObj:=wPaper;
    MoveL Offs(pOrigin,126.32,44.74,0.00),v40,z0,tPen\WObj:=wPaper;
    MoveL Offs(pOrigin,126.11,45.16,0.00),v40,z0,tPen\WObj:=wPaper;
    MoveL Offs(pOrigin,126.32,44.74,0.00),v40,z0,tPen\WObj:=wPaper;
    MoveL Offs(pOrigin,126.68,44.83,0.00),v40,z0,tPen\WObj:=wPaper;
    MoveL Offs(pOrigin,124.72,42.88,0.00),v40,z0,tPen\WObj:=wPaper;
    MoveL Offs(pOrigin,124.84,43.51,0.00),v40,z0,tPen\WObj:=wPaper;
    MoveL Offs(pOrigin,127.18,43.51,0.00),v40,z0,tPen\WObj:=wPaper;
    MoveL Offs(pOrigin,126.73,43.68,0.00),v40,z0,tPen\WObj:=wPaper;
    MoveL Offs(pOrigin,126.73,39.64,0.00),v40,z0,tPen\WObj:=wPaper;
    MoveL Offs(pOrigin,127.79,39.42,0.00),v40,z0,tPen\WObj:=wPaper;
    MoveL Offs(pOrigin,127.79,42.40,0.00),v40,z0,tPen\WObj:=wPaper;
    MoveL Offs(pOrigin,128.24,42.46,0.00),v40,z0,tPen\WObj:=wPaper;
    MoveL Offs(pOrigin,125.26,42.46,0.00),v40,z0,tPen\WObj:=wPaper;
    MoveL Offs(pOrigin,125.26,42.19,0.00),v40,z0,tPen\WObj:=wPaper;
    MoveL Offs(pOrigin,125.05,42.61,0.00),v40,z0,tPen\WObj:=wPaper;
    MoveL Offs(pOrigin,125.26,42.19,0.00),v40,z0,tPen\WObj:=wPaper;
    MoveL Offs(pOrigin,125.68,42.61,0.00),v40,z0,tPen\WObj:=wPaper;
    MoveL Offs(pOrigin,125.68,45.16,0.00),v40,z0,tPen\WObj:=wPaper;
    MoveL Offs(pOrigin,125.90,45.62,0.00),v40,z0,tPen\WObj:=wPaper;
    MoveL Offs(pOrigin,124.20,45.62,0.00),v40,z0,tPen\WObj:=wPaper;
    MoveL Offs(pOrigin,123.83,44.97,0.00),v40,z0,tPen\WObj:=wPaper;
    MoveL Offs(pOrigin,125.79,46.93,0.00),v40,z0,tPen\WObj:=wPaper;
    MoveL Offs(pOrigin,125.26,46.68,0.00),v40,z0,tPen\WObj:=wPaper;
    MoveL Offs(pOrigin,124.20,46.68,0.00),v40,z0,tPen\WObj:=wPaper;
    MoveL Offs(pOrigin,123.69,46.32,0.00),v40,z0,tPen\WObj:=wPaper;
    MoveL Offs(pOrigin,125.34,47.97,0.00),v40,fine,tPen\WObj:=wPaper;
    MoveL Offs(pOrigin,125.34,47.97,6.00),v60,z5,tPen\WObj:=wPaper;
    MoveL Offs(pOrigin,126.75,48.14,6.00),vTravel,z5,tPen\WObj:=wPaper;
    MoveL Offs(pOrigin,126.75,48.14,0.00),v60,z0,tPen\WObj:=wPaper;
    MoveL Offs(pOrigin,127.25,45.59,0.00),v40,z0,tPen\WObj:=wPaper;
    MoveL Offs(pOrigin,128.66,42.83,0.00),v40,z0,tPen\WObj:=wPaper;
    MoveL Offs(pOrigin,131.00,40.70,0.00),v40,z0,tPen\WObj:=wPaper;
    MoveL Offs(pOrigin,132.27,40.28,0.00),v40,z0,tPen\WObj:=wPaper;
    MoveL Offs(pOrigin,132.66,40.36,0.00),v40,z0,tPen\WObj:=wPaper;
    MoveL Offs(pOrigin,129.50,37.20,0.00),v40,z0,tPen\WObj:=wPaper;
    MoveL Offs(pOrigin,129.60,36.42,0.00),v40,z0,tPen\WObj:=wPaper;
    MoveL Offs(pOrigin,118.63,47.39,0.00),v40,z0,tPen\WObj:=wPaper;
    MoveL Offs(pOrigin,119.05,47.66,0.00),v40,z0,tPen\WObj:=wPaper;
    MoveL Offs(pOrigin,121.60,50.21,0.00),v40,z0,tPen\WObj:=wPaper;
    MoveL Offs(pOrigin,121.22,49.85,0.00),v40,z0,tPen\WObj:=wPaper;
    MoveL Offs(pOrigin,119.52,49.85,0.00),v40,z0,tPen\WObj:=wPaper;
    MoveL Offs(pOrigin,119.05,49.15,0.00),v40,z0,tPen\WObj:=wPaper;
    MoveL Offs(pOrigin,122.66,52.76,0.00),v40,z0,tPen\WObj:=wPaper;
    MoveL Offs(pOrigin,122.29,53.02,0.00),v40,z0,tPen\WObj:=wPaper;
    MoveL Offs(pOrigin,119.95,53.02,0.00),v40,z0,tPen\WObj:=wPaper;
    MoveL Offs(pOrigin,119.06,52.93,0.00),v40,z0,tPen\WObj:=wPaper;
    MoveL Offs(pOrigin,136.04,35.95,0.00),v40,z0,tPen\WObj:=wPaper;
    MoveL Offs(pOrigin,136.39,36.62,0.00),v40,z0,tPen\WObj:=wPaper;
    MoveL Offs(pOrigin,137.89,38.13,0.00),v40,z0,tPen\WObj:=wPaper;
    MoveL Offs(pOrigin,137.53,38.94,0.00),v40,z0,tPen\WObj:=wPaper;
    MoveL Offs(pOrigin,141.14,35.33,0.00),v40,z0,tPen\WObj:=wPaper;
    MoveL Offs(pOrigin,140.43,36.19,0.00),v40,z0,tPen\WObj:=wPaper;
    MoveL Offs(pOrigin,146.74,42.50,0.00),v40,z0,tPen\WObj:=wPaper;
  ENDPROC

  PROC DrawPart149()
    MoveL Offs(pOrigin,146.81,43.11,0.00),v40,z0,tPen\WObj:=wPaper;
    MoveL Offs(pOrigin,154.47,35.44,0.00),v40,fine,tPen\WObj:=wPaper;
    MoveL Offs(pOrigin,154.47,35.44,6.00),v60,z5,tPen\WObj:=wPaper;
    MoveL Offs(pOrigin,152.97,35.45,6.00),vTravel,z5,tPen\WObj:=wPaper;
    MoveL Offs(pOrigin,152.97,35.45,0.00),v60,z0,tPen\WObj:=wPaper;
    MoveL Offs(pOrigin,134.94,53.48,0.00),v40,z0,tPen\WObj:=wPaper;
    MoveL Offs(pOrigin,135.54,53.70,0.00),v40,z0,tPen\WObj:=wPaper;
    MoveL Offs(pOrigin,153.42,71.58,0.00),v40,z0,tPen\WObj:=wPaper;
    MoveL Offs(pOrigin,153.52,70.97,0.00),v40,z0,tPen\WObj:=wPaper;
    MoveL Offs(pOrigin,162.66,70.97,0.00),v40,z0,tPen\WObj:=wPaper;
    MoveL Offs(pOrigin,162.64,70.66,0.00),v40,z0,tPen\WObj:=wPaper;
    MoveL Offs(pOrigin,162.64,68.54,0.00),v40,z0,tPen\WObj:=wPaper;
    MoveL Offs(pOrigin,163.00,67.71,0.00),v40,z0,tPen\WObj:=wPaper;
    MoveL Offs(pOrigin,170.06,74.78,0.00),v40,z0,tPen\WObj:=wPaper;
    MoveL Offs(pOrigin,169.46,74.91,0.00),v40,z0,tPen\WObj:=wPaper;
    MoveL Offs(pOrigin,169.25,75.34,0.00),v40,z0,tPen\WObj:=wPaper;
    MoveL Offs(pOrigin,169.46,74.91,0.00),v40,fine,tPen\WObj:=wPaper;
    MoveL Offs(pOrigin,169.46,74.91,6.00),v60,z5,tPen\WObj:=wPaper;
    MoveL Offs(pOrigin,168.87,76.57,6.00),vTravel,z5,tPen\WObj:=wPaper;
    MoveL Offs(pOrigin,168.87,76.57,0.00),v60,z0,tPen\WObj:=wPaper;
    MoveL Offs(pOrigin,160.15,67.86,0.00),v40,z0,tPen\WObj:=wPaper;
    MoveL Offs(pOrigin,160.06,67.18,0.00),v40,z0,tPen\WObj:=wPaper;
    MoveL Offs(pOrigin,151.50,75.75,0.00),v40,z0,tPen\WObj:=wPaper;
    MoveL Offs(pOrigin,151.19,75.32,0.00),v40,z0,tPen\WObj:=wPaper;
    MoveL Offs(pOrigin,148.78,72.91,0.00),v40,z0,tPen\WObj:=wPaper;
    MoveL Offs(pOrigin,148.64,73.08,0.00),v40,z0,tPen\WObj:=wPaper;
    MoveL Offs(pOrigin,145.02,73.08,0.00),v40,fine,tPen\WObj:=wPaper;
    MoveL Offs(pOrigin,145.02,73.08,6.00),v60,z5,tPen\WObj:=wPaper;
    MoveL Offs(pOrigin,145.36,74.42,6.00),vTravel,z5,tPen\WObj:=wPaper;
    MoveL Offs(pOrigin,145.36,74.42,0.00),v60,z0,tPen\WObj:=wPaper;
    MoveL Offs(pOrigin,147.92,71.86,0.00),v40,z0,tPen\WObj:=wPaper;
    MoveL Offs(pOrigin,148.96,72.31,0.00),v40,z0,tPen\WObj:=wPaper;
    MoveL Offs(pOrigin,146.56,74.71,0.00),v40,fine,tPen\WObj:=wPaper;
    MoveL Offs(pOrigin,146.56,74.71,6.00),v60,z5,tPen\WObj:=wPaper;
    MoveL Offs(pOrigin,148.95,75.31,6.00),vTravel,z5,tPen\WObj:=wPaper;
    MoveL Offs(pOrigin,148.95,75.31,0.00),v60,z0,tPen\WObj:=wPaper;
    MoveL Offs(pOrigin,151.51,72.75,0.00),v40,z0,tPen\WObj:=wPaper;
    MoveL Offs(pOrigin,152.38,73.52,0.00),v40,z0,tPen\WObj:=wPaper;
    MoveL Offs(pOrigin,154.49,75.63,0.00),v40,fine,tPen\WObj:=wPaper;
    MoveL Offs(pOrigin,154.49,75.63,6.00),v60,z5,tPen\WObj:=wPaper;
    MoveL Offs(pOrigin,154.49,77.13,6.00),vTravel,z5,tPen\WObj:=wPaper;
    MoveL Offs(pOrigin,154.49,77.13,0.00),v60,z0,tPen\WObj:=wPaper;
    MoveL Offs(pOrigin,156.29,78.93,0.00),v40,z0,tPen\WObj:=wPaper;
    MoveL Offs(pOrigin,155.65,78.36,0.00),v40,z0,tPen\WObj:=wPaper;
    MoveL Offs(pOrigin,152.04,78.36,0.00),v40,z0,tPen\WObj:=wPaper;
    MoveL Offs(pOrigin,152.24,77.87,0.00),v40,z0,tPen\WObj:=wPaper;
    MoveL Offs(pOrigin,154.05,79.67,0.00),v40,z0,tPen\WObj:=wPaper;
    MoveL Offs(pOrigin,154.78,79.93,0.00),v40,z0,tPen\WObj:=wPaper;
    MoveL Offs(pOrigin,167.85,66.86,0.00),v40,z0,tPen\WObj:=wPaper;
    MoveL Offs(pOrigin,168.40,65.99,0.00),v40,z0,tPen\WObj:=wPaper;
    MoveL Offs(pOrigin,167.76,65.56,0.00),v40,z0,tPen\WObj:=wPaper;
    MoveL Offs(pOrigin,165.71,62.59,0.00),v40,z0,tPen\WObj:=wPaper;
    MoveL Offs(pOrigin,165.00,60.89,0.00),v40,fine,tPen\WObj:=wPaper;
    MoveL Offs(pOrigin,165.00,60.89,6.00),v60,z5,tPen\WObj:=wPaper;
    MoveL Offs(pOrigin,166.27,67.69,6.00),vTravel,z5,tPen\WObj:=wPaper;
    MoveL Offs(pOrigin,166.27,67.69,0.00),v60,z0,tPen\WObj:=wPaper;
    MoveL Offs(pOrigin,165.64,68.11,0.00),v40,z0,tPen\WObj:=wPaper;
    MoveL Offs(pOrigin,158.62,67.90,0.00),v40,z0,tPen\WObj:=wPaper;
    MoveL Offs(pOrigin,155.23,66.77,0.00),v40,z0,tPen\WObj:=wPaper;
    MoveL Offs(pOrigin,152.25,64.93,0.00),v40,z0,tPen\WObj:=wPaper;
    MoveL Offs(pOrigin,151.82,63.86,0.00),v40,z0,tPen\WObj:=wPaper;
    MoveL Offs(pOrigin,148.64,60.46,0.00),v40,z0,tPen\WObj:=wPaper;
    MoveL Offs(pOrigin,146.94,57.91,0.00),v40,z0,tPen\WObj:=wPaper;
    MoveL Offs(pOrigin,146.94,57.91,0.00),v40,z0,tPen\WObj:=wPaper;
    MoveL Offs(pOrigin,145.59,56.85,0.00),v40,z0,tPen\WObj:=wPaper;
    MoveL Offs(pOrigin,143.96,52.81,0.00),v40,z0,tPen\WObj:=wPaper;
    MoveL Offs(pOrigin,143.32,50.26,0.00),v40,z0,tPen\WObj:=wPaper;
    MoveL Offs(pOrigin,143.61,46.22,0.00),v40,z0,tPen\WObj:=wPaper;
    MoveL Offs(pOrigin,144.32,45.52,0.00),v40,z0,tPen\WObj:=wPaper;
    MoveL Offs(pOrigin,144.60,44.31,0.00),v40,z0,tPen\WObj:=wPaper;
    MoveL Offs(pOrigin,147.15,42.12,0.00),v40,z0,tPen\WObj:=wPaper;
    MoveL Offs(pOrigin,152.68,40.35,0.00),v40,z0,tPen\WObj:=wPaper;
    MoveL Offs(pOrigin,155.23,38.79,0.00),v40,fine,tPen\WObj:=wPaper;
    MoveL Offs(pOrigin,155.23,38.79,6.00),v60,z5,tPen\WObj:=wPaper;
    MoveL Offs(pOrigin,156.70,39.18,6.00),vTravel,z5,tPen\WObj:=wPaper;
    MoveL Offs(pOrigin,156.70,39.18,0.00),v60,z0,tPen\WObj:=wPaper;
    MoveL Offs(pOrigin,164.67,31.22,0.00),v40,z0,tPen\WObj:=wPaper;
    MoveL Offs(pOrigin,164.69,32.07,0.00),v40,z0,tPen\WObj:=wPaper;
    MoveL Offs(pOrigin,166.19,33.57,0.00),v40,z0,tPen\WObj:=wPaper;
    MoveL Offs(pOrigin,166.61,33.76,0.00),v40,z0,tPen\WObj:=wPaper;
    MoveL Offs(pOrigin,169.76,30.60,0.00),v40,z0,tPen\WObj:=wPaper;
    MoveL Offs(pOrigin,170.08,31.48,0.00),v40,z0,tPen\WObj:=wPaper;
    MoveL Offs(pOrigin,171.58,32.99,0.00),v40,z0,tPen\WObj:=wPaper;
    MoveL Offs(pOrigin,171.40,33.44,0.00),v40,z0,tPen\WObj:=wPaper;
    MoveL Offs(pOrigin,174.11,30.74,0.00),v40,z0,tPen\WObj:=wPaper;
    MoveL Offs(pOrigin,174.27,31.20,0.00),v40,z0,tPen\WObj:=wPaper;
    MoveL Offs(pOrigin,176.53,33.45,0.00),v40,fine,tPen\WObj:=wPaper;
    MoveL Offs(pOrigin,176.53,33.45,6.00),v60,z5,tPen\WObj:=wPaper;
    MoveL Offs(pOrigin,174.56,33.90,6.00),vTravel,z5,tPen\WObj:=wPaper;
    MoveL Offs(pOrigin,174.56,33.90,0.00),v60,z0,tPen\WObj:=wPaper;
    MoveL Offs(pOrigin,175.62,33.62,0.00),v40,z0,tPen\WObj:=wPaper;
    MoveL Offs(pOrigin,176.26,33.05,0.00),v40,z0,tPen\WObj:=wPaper;
    MoveL Offs(pOrigin,180.73,32.62,0.00),v40,z0,tPen\WObj:=wPaper;
    MoveL Offs(pOrigin,190.50,32.41,0.00),v40,z0,tPen\WObj:=wPaper;
    MoveL Offs(pOrigin,195.81,33.26,0.00),v40,z0,tPen\WObj:=wPaper;
    MoveL Offs(pOrigin,198.15,34.25,0.00),v40,z0,tPen\WObj:=wPaper;
    MoveL Offs(pOrigin,199.28,35.17,0.00),v40,z0,tPen\WObj:=wPaper;
    MoveL Offs(pOrigin,199.00,35.60,0.00),v40,z0,tPen\WObj:=wPaper;
    MoveL Offs(pOrigin,195.60,35.60,0.00),v40,z0,tPen\WObj:=wPaper;
    MoveL Offs(pOrigin,193.05,36.03,0.00),v40,z0,tPen\WObj:=wPaper;
    MoveL Offs(pOrigin,188.59,37.30,0.00),v40,z0,tPen\WObj:=wPaper;
    MoveL Offs(pOrigin,187.52,37.30,0.00),v40,z0,tPen\WObj:=wPaper;
    MoveL Offs(pOrigin,186.25,37.94,0.00),v40,z0,tPen\WObj:=wPaper;
    MoveL Offs(pOrigin,186.57,37.53,0.00),v40,z0,tPen\WObj:=wPaper;
    MoveL Offs(pOrigin,188.38,39.33,0.00),v40,z0,tPen\WObj:=wPaper;
    MoveL Offs(pOrigin,188.76,39.98,0.00),v40,z0,tPen\WObj:=wPaper;
    MoveL Offs(pOrigin,193.87,34.87,0.00),v40,fine,tPen\WObj:=wPaper;
    MoveL Offs(pOrigin,193.87,34.87,6.00),v60,z5,tPen\WObj:=wPaper;
    MoveL Offs(pOrigin,193.57,33.68,6.00),vTravel,z5,tPen\WObj:=wPaper;
    MoveL Offs(pOrigin,193.57,33.68,0.00),v60,z0,tPen\WObj:=wPaper;
    MoveL Offs(pOrigin,196.28,30.97,0.00),v40,fine,tPen\WObj:=wPaper;
    MoveL Offs(pOrigin,196.28,30.97,6.00),v60,z5,tPen\WObj:=wPaper;
    MoveL Offs(pOrigin,198.52,31.71,6.00),vTravel,z5,tPen\WObj:=wPaper;
    MoveL Offs(pOrigin,198.52,31.71,0.00),v60,z0,tPen\WObj:=wPaper;
    MoveL Offs(pOrigin,189.51,40.73,0.00),v40,z0,tPen\WObj:=wPaper;
    MoveL Offs(pOrigin,190.50,40.06,0.00),v40,z0,tPen\WObj:=wPaper;
    MoveL Offs(pOrigin,190.29,41.12,0.00),v40,z0,tPen\WObj:=wPaper;
    MoveL Offs(pOrigin,190.50,41.55,0.00),v40,z0,tPen\WObj:=wPaper;
    MoveL Offs(pOrigin,190.93,41.55,0.00),v40,z0,tPen\WObj:=wPaper;
    MoveL Offs(pOrigin,191.14,40.49,0.00),v40,fine,tPen\WObj:=wPaper;
  ENDPROC

  PROC DrawPart150()
    MoveL Offs(pOrigin,191.14,40.49,6.00),v60,z5,tPen\WObj:=wPaper;
    MoveL Offs(pOrigin,192.21,39.52,6.00),vTravel,z5,tPen\WObj:=wPaper;
    MoveL Offs(pOrigin,192.21,39.52,0.00),v60,z0,tPen\WObj:=wPaper;
    MoveL Offs(pOrigin,186.20,45.53,0.00),v40,z0,tPen\WObj:=wPaper;
    MoveL Offs(pOrigin,185.30,44.94,0.00),v40,z0,tPen\WObj:=wPaper;
    MoveL Offs(pOrigin,187.25,42.98,0.00),v40,z0,tPen\WObj:=wPaper;
    MoveL Offs(pOrigin,186.51,42.24,0.00),v40,z0,tPen\WObj:=wPaper;
    MoveL Offs(pOrigin,184.55,44.19,0.00),v40,z0,tPen\WObj:=wPaper;
    MoveL Offs(pOrigin,183.96,43.29,0.00),v40,z0,tPen\WObj:=wPaper;
    MoveL Offs(pOrigin,191.77,35.48,0.00),v40,z0,tPen\WObj:=wPaper;
    MoveL Offs(pOrigin,191.21,36.19,0.00),v40,z0,tPen\WObj:=wPaper;
    MoveL Offs(pOrigin,192.87,37.85,0.00),v40,z0,tPen\WObj:=wPaper;
    MoveL Offs(pOrigin,192.20,37.18,0.00),v40,z0,tPen\WObj:=wPaper;
    MoveL Offs(pOrigin,188.59,37.18,0.00),v40,z0,tPen\WObj:=wPaper;
    MoveL Offs(pOrigin,188.97,36.94,0.00),v40,z0,tPen\WObj:=wPaper;
    MoveL Offs(pOrigin,191.07,39.04,0.00),v40,fine,tPen\WObj:=wPaper;
    MoveL Offs(pOrigin,191.07,39.04,6.00),v60,z5,tPen\WObj:=wPaper;
    MoveL Offs(pOrigin,193.86,37.87,6.00),vTravel,z5,tPen\WObj:=wPaper;
    MoveL Offs(pOrigin,193.86,37.87,0.00),v60,z0,tPen\WObj:=wPaper;
    MoveL Offs(pOrigin,199.72,32.01,0.00),v40,fine,tPen\WObj:=wPaper;
    MoveL Offs(pOrigin,199.72,32.01,6.00),v60,z5,tPen\WObj:=wPaper;
    MoveL Offs(pOrigin,199.60,33.47,6.00),vTravel,z5,tPen\WObj:=wPaper;
    MoveL Offs(pOrigin,199.60,33.47,0.00),v60,z0,tPen\WObj:=wPaper;
    MoveL Offs(pOrigin,199.60,36.45,0.00),v40,fine,tPen\WObj:=wPaper;
    MoveL Offs(pOrigin,199.60,36.45,6.00),v60,z5,tPen\WObj:=wPaper;
    MoveL Offs(pOrigin,201.71,36.88,6.00),vTravel,z5,tPen\WObj:=wPaper;
    MoveL Offs(pOrigin,201.71,36.88,0.00),v60,z0,tPen\WObj:=wPaper;
    MoveL Offs(pOrigin,201.71,35.17,0.00),v40,fine,tPen\WObj:=wPaper;
    MoveL Offs(pOrigin,201.71,35.17,6.00),v60,z5,tPen\WObj:=wPaper;
    MoveL Offs(pOrigin,204.63,42.03,6.00),vTravel,z5,tPen\WObj:=wPaper;
    MoveL Offs(pOrigin,204.63,42.03,0.00),v60,z0,tPen\WObj:=wPaper;
    MoveL Offs(pOrigin,200.27,46.39,0.00),v40,z0,tPen\WObj:=wPaper;
    MoveL Offs(pOrigin,199.63,46.11,0.00),v40,z0,tPen\WObj:=wPaper;
    MoveL Offs(pOrigin,198.28,44.75,0.00),v40,z0,tPen\WObj:=wPaper;
    MoveL Offs(pOrigin,198.18,44.00,0.00),v40,z0,tPen\WObj:=wPaper;
    MoveL Offs(pOrigin,193.98,48.20,0.00),v40,z0,tPen\WObj:=wPaper;
    MoveL Offs(pOrigin,193.80,47.74,0.00),v40,z0,tPen\WObj:=wPaper;
    MoveL Offs(pOrigin,192.44,46.38,0.00),v40,fine,tPen\WObj:=wPaper;
    MoveL Offs(pOrigin,192.44,46.38,6.00),v60,z5,tPen\WObj:=wPaper;
    MoveL Offs(pOrigin,194.84,45.79,6.00),vTravel,z5,tPen\WObj:=wPaper;
    MoveL Offs(pOrigin,194.84,45.79,0.00),v60,z0,tPen\WObj:=wPaper;
    MoveL Offs(pOrigin,196.19,47.14,0.00),v40,z0,tPen\WObj:=wPaper;
    MoveL Offs(pOrigin,196.08,47.60,0.00),v40,z0,tPen\WObj:=wPaper;
    MoveL Offs(pOrigin,200.43,43.24,0.00),v40,z0,tPen\WObj:=wPaper;
    MoveL Offs(pOrigin,200.68,44.16,0.00),v40,z0,tPen\WObj:=wPaper;
    MoveL Offs(pOrigin,202.03,45.51,0.00),v40,z0,tPen\WObj:=wPaper;
    MoveL Offs(pOrigin,202.22,45.93,0.00),v40,z0,tPen\WObj:=wPaper;
    MoveL Offs(pOrigin,209.29,38.87,0.00),v40,fine,tPen\WObj:=wPaper;
    MoveL Offs(pOrigin,209.29,38.87,6.00),v60,z5,tPen\WObj:=wPaper;
    MoveL Offs(pOrigin,209.41,40.28,6.00),vTravel,z5,tPen\WObj:=wPaper;
    MoveL Offs(pOrigin,209.41,40.28,0.00),v60,z0,tPen\WObj:=wPaper;
    MoveL Offs(pOrigin,209.62,40.70,0.00),v40,z0,tPen\WObj:=wPaper;
    MoveL Offs(pOrigin,209.41,40.28,0.00),v40,z0,tPen\WObj:=wPaper;
    MoveL Offs(pOrigin,209.10,40.70,0.00),v40,z0,tPen\WObj:=wPaper;
    MoveL Offs(pOrigin,209.10,42.82,0.00),v40,z0,tPen\WObj:=wPaper;
    MoveL Offs(pOrigin,209.21,43.74,0.00),v40,z0,tPen\WObj:=wPaper;
    MoveL Offs(pOrigin,207.26,41.78,0.00),v40,z0,tPen\WObj:=wPaper;
    MoveL Offs(pOrigin,207.08,42.46,0.00),v40,z0,tPen\WObj:=wPaper;
    MoveL Offs(pOrigin,215.15,42.46,0.00),v40,z0,tPen\WObj:=wPaper;
    MoveL Offs(pOrigin,214.58,42.40,0.00),v40,z0,tPen\WObj:=wPaper;
    MoveL Offs(pOrigin,214.58,42.83,0.00),v40,z0,tPen\WObj:=wPaper;
    MoveL Offs(pOrigin,216.07,44.74,0.00),v40,z0,tPen\WObj:=wPaper;
    MoveL Offs(pOrigin,216.64,46.30,0.00),v40,z0,tPen\WObj:=wPaper;
    MoveL Offs(pOrigin,217.49,46.08,0.00),v40,z0,tPen\WObj:=wPaper;
    MoveL Offs(pOrigin,218.48,45.30,0.00),v40,z0,tPen\WObj:=wPaper;
    MoveL Offs(pOrigin,217.42,42.26,0.00),v40,z0,tPen\WObj:=wPaper;
    MoveL Offs(pOrigin,214.58,42.40,0.00),v40,z0,tPen\WObj:=wPaper;
    MoveL Offs(pOrigin,214.38,41.55,0.00),v40,z0,tPen\WObj:=wPaper;
    MoveL Offs(pOrigin,214.38,43.89,0.00),v40,z0,tPen\WObj:=wPaper;
    MoveL Offs(pOrigin,213.88,44.31,0.00),v40,z0,tPen\WObj:=wPaper;
    MoveL Offs(pOrigin,214.51,44.95,0.00),v40,z0,tPen\WObj:=wPaper;
    MoveL Offs(pOrigin,213.88,44.31,0.00),v40,z0,tPen\WObj:=wPaper;
    MoveL Offs(pOrigin,214.51,44.57,0.00),v40,z0,tPen\WObj:=wPaper;
    MoveL Offs(pOrigin,216.00,44.57,0.00),v40,z0,tPen\WObj:=wPaper;
    MoveL Offs(pOrigin,216.00,44.31,0.00),v40,z0,tPen\WObj:=wPaper;
    MoveL Offs(pOrigin,216.21,44.74,0.00),v40,z0,tPen\WObj:=wPaper;
    MoveL Offs(pOrigin,216.00,44.31,0.00),v40,z0,tPen\WObj:=wPaper;
    MoveL Offs(pOrigin,215.36,43.51,0.00),v40,z0,tPen\WObj:=wPaper;
    MoveL Offs(pOrigin,213.02,43.51,0.00),v40,z0,tPen\WObj:=wPaper;
    MoveL Offs(pOrigin,213.33,43.46,0.00),v40,z0,tPen\WObj:=wPaper;
    MoveL Offs(pOrigin,213.33,41.34,0.00),v40,z0,tPen\WObj:=wPaper;
    MoveL Offs(pOrigin,213.55,40.61,0.00),v40,z0,tPen\WObj:=wPaper;
    MoveL Offs(pOrigin,215.95,43.01,0.00),v40,z0,tPen\WObj:=wPaper;
    MoveL Offs(pOrigin,215.15,43.25,0.00),v40,z0,tPen\WObj:=wPaper;
    MoveL Offs(pOrigin,215.57,43.67,0.00),v40,z0,tPen\WObj:=wPaper;
    MoveL Offs(pOrigin,215.15,43.25,0.00),v40,fine,tPen\WObj:=wPaper;
    MoveL Offs(pOrigin,215.15,43.25,6.00),v60,z5,tPen\WObj:=wPaper;
    MoveL Offs(pOrigin,217.28,42.46,6.00),vTravel,z5,tPen\WObj:=wPaper;
    MoveL Offs(pOrigin,217.28,42.46,0.00),v60,z0,tPen\WObj:=wPaper;
    MoveL Offs(pOrigin,219.61,42.46,0.00),v40,z0,tPen\WObj:=wPaper;
    MoveL Offs(pOrigin,220.04,43.51,0.00),v40,z0,tPen\WObj:=wPaper;
    MoveL Offs(pOrigin,218.12,43.51,0.00),v40,z0,tPen\WObj:=wPaper;
    MoveL Offs(pOrigin,218.34,44.57,0.00),v40,z0,tPen\WObj:=wPaper;
    MoveL Offs(pOrigin,222.16,44.57,0.00),v40,z0,tPen\WObj:=wPaper;
    MoveL Offs(pOrigin,221.95,45.16,0.00),v40,z0,tPen\WObj:=wPaper;
    MoveL Offs(pOrigin,221.10,45.16,0.00),v40,z0,tPen\WObj:=wPaper;
    MoveL Offs(pOrigin,220.68,46.01,0.00),v40,z0,tPen\WObj:=wPaper;
    MoveL Offs(pOrigin,220.46,45.62,0.00),v40,z0,tPen\WObj:=wPaper;
    MoveL Offs(pOrigin,214.94,45.62,0.00),v40,z0,tPen\WObj:=wPaper;
    MoveL Offs(pOrigin,215.44,45.59,0.00),v40,z0,tPen\WObj:=wPaper;
    MoveL Offs(pOrigin,215.44,48.99,0.00),v40,z0,tPen\WObj:=wPaper;
    MoveL Offs(pOrigin,216.42,49.45,0.00),v40,z0,tPen\WObj:=wPaper;
    MoveL Offs(pOrigin,214.47,47.50,0.00),v40,z0,tPen\WObj:=wPaper;
    MoveL Offs(pOrigin,214.94,47.74,0.00),v40,z0,tPen\WObj:=wPaper;
    MoveL Offs(pOrigin,217.49,47.74,0.00),v40,z0,tPen\WObj:=wPaper;
    MoveL Offs(pOrigin,217.70,48.14,0.00),v40,z0,tPen\WObj:=wPaper;
    MoveL Offs(pOrigin,216.85,48.35,0.00),v40,z0,tPen\WObj:=wPaper;
    MoveL Offs(pOrigin,216.64,48.99,0.00),v40,z0,tPen\WObj:=wPaper;
    MoveL Offs(pOrigin,217.49,49.06,0.00),v40,z0,tPen\WObj:=wPaper;
    MoveL Offs(pOrigin,217.91,48.35,0.00),v40,z0,tPen\WObj:=wPaper;
    MoveL Offs(pOrigin,217.91,48.35,0.00),v40,z0,tPen\WObj:=wPaper;
    MoveL Offs(pOrigin,218.55,48.14,0.00),v40,z0,tPen\WObj:=wPaper;
    MoveL Offs(pOrigin,218.98,47.50,0.00),v40,z0,tPen\WObj:=wPaper;
    MoveL Offs(pOrigin,218.76,47.29,0.00),v40,z0,tPen\WObj:=wPaper;
    MoveL Offs(pOrigin,219.19,47.08,0.00),v40,z0,tPen\WObj:=wPaper;
    MoveL Offs(pOrigin,218.96,47.51,0.00),v40,z0,tPen\WObj:=wPaper;
    MoveL Offs(pOrigin,212.20,40.75,0.00),v40,z0,tPen\WObj:=wPaper;
    MoveL Offs(pOrigin,212.27,41.34,0.00),v40,z0,tPen\WObj:=wPaper;
    MoveL Offs(pOrigin,212.27,43.04,0.00),v40,z0,tPen\WObj:=wPaper;
    MoveL Offs(pOrigin,211.21,42.82,0.00),v40,z0,tPen\WObj:=wPaper;
  ENDPROC

  PROC DrawPart151()
    MoveL Offs(pOrigin,211.21,41.55,0.00),v40,z0,tPen\WObj:=wPaper;
    MoveL Offs(pOrigin,210.70,40.75,0.00),v40,z0,tPen\WObj:=wPaper;
    MoveL Offs(pOrigin,218.07,48.11,0.00),v40,z0,tPen\WObj:=wPaper;
    MoveL Offs(pOrigin,217.70,48.14,0.00),v40,z0,tPen\WObj:=wPaper;
    MoveL Offs(pOrigin,218.12,47.29,0.00),v40,z0,tPen\WObj:=wPaper;
    MoveL Offs(pOrigin,218.55,47.29,0.00),v40,z0,tPen\WObj:=wPaper;
    MoveL Offs(pOrigin,218.76,46.68,0.00),v40,z0,tPen\WObj:=wPaper;
    MoveL Offs(pOrigin,215.15,46.68,0.00),v40,z0,tPen\WObj:=wPaper;
    MoveL Offs(pOrigin,214.46,46.00,0.00),v40,z0,tPen\WObj:=wPaper;
    MoveL Offs(pOrigin,217.17,48.71,0.00),v40,z0,tPen\WObj:=wPaper;
    MoveL Offs(pOrigin,216.49,47.92,0.00),v40,z0,tPen\WObj:=wPaper;
    MoveL Offs(pOrigin,216.49,46.22,0.00),v40,fine,tPen\WObj:=wPaper;
    MoveL Offs(pOrigin,216.49,46.22,6.00),v60,z5,tPen\WObj:=wPaper;
    MoveL Offs(pOrigin,217.61,44.66,6.00),vTravel,z5,tPen\WObj:=wPaper;
    MoveL Offs(pOrigin,217.61,44.66,0.00),v60,z0,tPen\WObj:=wPaper;
    MoveL Offs(pOrigin,219.86,46.92,0.00),v40,fine,tPen\WObj:=wPaper;
    MoveL Offs(pOrigin,219.86,46.92,6.00),v60,z5,tPen\WObj:=wPaper;
    MoveL Offs(pOrigin,219.66,45.59,6.00),vTravel,z5,tPen\WObj:=wPaper;
    MoveL Offs(pOrigin,219.66,45.59,0.00),v60,z0,tPen\WObj:=wPaper;
    MoveL Offs(pOrigin,219.66,44.10,0.00),v40,fine,tPen\WObj:=wPaper;
    MoveL Offs(pOrigin,219.66,44.10,6.00),v60,z5,tPen\WObj:=wPaper;
    MoveL Offs(pOrigin,221.31,43.67,6.00),vTravel,z5,tPen\WObj:=wPaper;
    MoveL Offs(pOrigin,221.31,43.67,0.00),v60,z0,tPen\WObj:=wPaper;
    MoveL Offs(pOrigin,220.04,44.17,0.00),v40,z0,tPen\WObj:=wPaper;
    MoveL Offs(pOrigin,219.26,42.83,0.00),v40,z0,tPen\WObj:=wPaper;
    MoveL Offs(pOrigin,219.26,42.05,0.00),v40,z0,tPen\WObj:=wPaper;
    MoveL Offs(pOrigin,223.23,41.55,0.00),v40,z0,tPen\WObj:=wPaper;
    MoveL Offs(pOrigin,224.50,41.76,0.00),v40,z0,tPen\WObj:=wPaper;
    MoveL Offs(pOrigin,224.50,41.76,0.00),v40,z0,tPen\WObj:=wPaper;
    MoveL Offs(pOrigin,224.85,43.46,0.00),v40,z0,tPen\WObj:=wPaper;
    MoveL Offs(pOrigin,223.23,44.95,0.00),v40,z0,tPen\WObj:=wPaper;
    MoveL Offs(pOrigin,223.44,44.57,0.00),v40,z0,tPen\WObj:=wPaper;
    MoveL Offs(pOrigin,225.56,44.57,0.00),v40,z0,tPen\WObj:=wPaper;
    MoveL Offs(pOrigin,225.35,44.95,0.00),v40,z0,tPen\WObj:=wPaper;
    MoveL Offs(pOrigin,224.93,45.59,0.00),v40,z0,tPen\WObj:=wPaper;
    MoveL Offs(pOrigin,225.35,44.95,0.00),v40,z0,tPen\WObj:=wPaper;
    MoveL Offs(pOrigin,225.70,45.29,0.00),v40,z0,tPen\WObj:=wPaper;
    MoveL Offs(pOrigin,220.59,40.18,0.00),v40,z0,tPen\WObj:=wPaper;
    MoveL Offs(pOrigin,220.52,39.58,0.00),v40,z0,tPen\WObj:=wPaper;
    MoveL Offs(pOrigin,214.06,46.05,0.00),v40,z0,tPen\WObj:=wPaper;
    MoveL Offs(pOrigin,213.46,45.15,0.00),v40,z0,tPen\WObj:=wPaper;
    MoveL Offs(pOrigin,219.02,39.59,0.00),v40,fine,tPen\WObj:=wPaper;
    MoveL Offs(pOrigin,219.02,39.59,6.00),v60,z5,tPen\WObj:=wPaper;
    MoveL Offs(pOrigin,218.61,40.91,6.00),vTravel,z5,tPen\WObj:=wPaper;
    MoveL Offs(pOrigin,218.61,40.91,0.00),v60,z0,tPen\WObj:=wPaper;
    MoveL Offs(pOrigin,218.61,46.22,0.00),v40,fine,tPen\WObj:=wPaper;
    MoveL Offs(pOrigin,218.61,46.22,6.00),v60,z5,tPen\WObj:=wPaper;
    MoveL Offs(pOrigin,219.86,48.41,6.00),vTravel,z5,tPen\WObj:=wPaper;
    MoveL Offs(pOrigin,219.86,48.41,0.00),v60,z0,tPen\WObj:=wPaper;
    MoveL Offs(pOrigin,223.62,52.17,0.00),v40,z0,tPen\WObj:=wPaper;
    MoveL Offs(pOrigin,224.07,52.46,0.00),v40,z0,tPen\WObj:=wPaper;
    MoveL Offs(pOrigin,221.67,54.86,0.00),v40,z0,tPen\WObj:=wPaper;
    MoveL Offs(pOrigin,222.13,55.16,0.00),v40,z0,tPen\WObj:=wPaper;
    MoveL Offs(pOrigin,225.74,58.77,0.00),v40,z0,tPen\WObj:=wPaper;
    MoveL Offs(pOrigin,225.85,58.14,0.00),v40,z0,tPen\WObj:=wPaper;
    MoveL Offs(pOrigin,223.30,60.70,0.00),v40,z0,tPen\WObj:=wPaper;
    MoveL Offs(pOrigin,223.95,61.46,0.00),v40,z0,tPen\WObj:=wPaper;
    MoveL Offs(pOrigin,228.16,65.67,0.00),v40,z0,tPen\WObj:=wPaper;
    MoveL Offs(pOrigin,227.26,65.69,0.00),v40,z0,tPen\WObj:=wPaper;
    MoveL Offs(pOrigin,225.78,65.69,0.00),v40,z0,tPen\WObj:=wPaper;
    MoveL Offs(pOrigin,226.00,65.78,0.00),v40,z0,tPen\WObj:=wPaper;
    MoveL Offs(pOrigin,226.00,64.07,0.00),v40,z0,tPen\WObj:=wPaper;
    MoveL Offs(pOrigin,226.62,63.58,0.00),v40,z0,tPen\WObj:=wPaper;
    MoveL Offs(pOrigin,225.14,63.58,0.00),v40,z0,tPen\WObj:=wPaper;
    MoveL Offs(pOrigin,224.40,63.41,0.00),v40,z0,tPen\WObj:=wPaper;
    MoveL Offs(pOrigin,228.46,67.47,0.00),v40,z0,tPen\WObj:=wPaper;
    MoveL Offs(pOrigin,227.69,67.80,0.00),v40,z0,tPen\WObj:=wPaper;
    MoveL Offs(pOrigin,226.20,67.80,0.00),v40,z0,tPen\WObj:=wPaper;
    MoveL Offs(pOrigin,225.23,67.73,0.00),v40,z0,tPen\WObj:=wPaper;
    MoveL Offs(pOrigin,230.63,62.32,0.00),v40,fine,tPen\WObj:=wPaper;
    MoveL Offs(pOrigin,230.63,62.32,6.00),v60,z5,tPen\WObj:=wPaper;
    MoveL Offs(pOrigin,231.83,64.12,6.00),vTravel,z5,tPen\WObj:=wPaper;
    MoveL Offs(pOrigin,231.83,64.12,0.00),v60,z0,tPen\WObj:=wPaper;
    MoveL Offs(pOrigin,225.67,70.28,0.00),v40,z0,tPen\WObj:=wPaper;
    MoveL Offs(pOrigin,225.92,69.41,0.00),v40,z0,tPen\WObj:=wPaper;
    MoveL Offs(pOrigin,229.23,72.71,0.00),v40,z0,tPen\WObj:=wPaper;
    MoveL Offs(pOrigin,229.56,72.36,0.00),v40,z0,tPen\WObj:=wPaper;
    MoveL Offs(pOrigin,226.85,75.07,0.00),v40,z0,tPen\WObj:=wPaper;
    MoveL Offs(pOrigin,227.14,75.10,0.00),v40,z0,tPen\WObj:=wPaper;
    MoveL Offs(pOrigin,230.29,78.26,0.00),v40,z0,tPen\WObj:=wPaper;
    MoveL Offs(pOrigin,229.81,78.36,0.00),v40,z0,tPen\WObj:=wPaper;
    MoveL Offs(pOrigin,228.54,78.36,0.00),v40,z0,tPen\WObj:=wPaper;
    MoveL Offs(pOrigin,227.90,78.85,0.00),v40,z0,tPen\WObj:=wPaper;
    MoveL Offs(pOrigin,231.50,82.45,0.00),v40,z0,tPen\WObj:=wPaper;
    MoveL Offs(pOrigin,230.88,82.58,0.00),v40,z0,tPen\WObj:=wPaper;
    MoveL Offs(pOrigin,229.18,82.58,0.00),v40,z0,tPen\WObj:=wPaper;
    MoveL Offs(pOrigin,228.51,82.45,0.00),v40,z0,tPen\WObj:=wPaper;
    MoveL Offs(pOrigin,231.36,85.30,0.00),v40,z0,tPen\WObj:=wPaper;
    MoveL Offs(pOrigin,231.76,85.09,0.00),v40,z0,tPen\WObj:=wPaper;
    MoveL Offs(pOrigin,228.91,87.94,0.00),v40,z0,tPen\WObj:=wPaper;
    MoveL Offs(pOrigin,228.97,87.39,0.00),v40,z0,tPen\WObj:=wPaper;
    MoveL Offs(pOrigin,231.83,90.25,0.00),v40,z0,tPen\WObj:=wPaper;
    MoveL Offs(pOrigin,232.35,90.48,0.00),v40,z0,tPen\WObj:=wPaper;
    MoveL Offs(pOrigin,229.49,93.33,0.00),v40,z0,tPen\WObj:=wPaper;
    MoveL Offs(pOrigin,230.45,93.14,0.00),v40,z0,tPen\WObj:=wPaper;
    MoveL Offs(pOrigin,231.72,93.14,0.00),v40,z0,tPen\WObj:=wPaper;
    MoveL Offs(pOrigin,232.29,93.69,0.00),v40,z0,tPen\WObj:=wPaper;
    MoveL Offs(pOrigin,229.43,90.84,0.00),v40,z0,tPen\WObj:=wPaper;
    MoveL Offs(pOrigin,229.05,90.79,0.00),v40,z0,tPen\WObj:=wPaper;
    MoveL Offs(pOrigin,232.05,87.78,0.00),v40,z0,tPen\WObj:=wPaper;
    MoveL Offs(pOrigin,231.09,87.86,0.00),v40,z0,tPen\WObj:=wPaper;
    MoveL Offs(pOrigin,229.81,87.86,0.00),v40,z0,tPen\WObj:=wPaper;
    MoveL Offs(pOrigin,229.81,86.81,0.00),v40,z0,tPen\WObj:=wPaper;
    MoveL Offs(pOrigin,230.88,86.81,0.00),v40,z0,tPen\WObj:=wPaper;
    MoveL Offs(pOrigin,231.52,86.95,0.00),v40,z0,tPen\WObj:=wPaper;
    MoveL Offs(pOrigin,228.66,84.09,0.00),v40,z0,tPen\WObj:=wPaper;
    MoveL Offs(pOrigin,228.32,84.05,0.00),v40,z0,tPen\WObj:=wPaper;
    MoveL Offs(pOrigin,234.48,77.89,0.00),v40,fine,tPen\WObj:=wPaper;
    MoveL Offs(pOrigin,234.48,77.89,6.00),v60,z5,tPen\WObj:=wPaper;
    MoveL Offs(pOrigin,233.21,77.89,6.00),vTravel,z5,tPen\WObj:=wPaper;
    MoveL Offs(pOrigin,233.21,77.89,0.00),v60,z0,tPen\WObj:=wPaper;
    MoveL Offs(pOrigin,233.00,78.31,0.00),v40,z0,tPen\WObj:=wPaper;
    MoveL Offs(pOrigin,233.21,77.89,0.00),v40,fine,tPen\WObj:=wPaper;
    MoveL Offs(pOrigin,233.21,77.89,6.00),v60,z5,tPen\WObj:=wPaper;
    MoveL Offs(pOrigin,232.57,78.95,6.00),vTravel,z5,tPen\WObj:=wPaper;
    MoveL Offs(pOrigin,232.57,78.95,0.00),v60,z0,tPen\WObj:=wPaper;
    MoveL Offs(pOrigin,232.36,79.38,0.00),v40,z0,tPen\WObj:=wPaper;
    MoveL Offs(pOrigin,232.57,78.95,0.00),v40,fine,tPen\WObj:=wPaper;
    MoveL Offs(pOrigin,232.57,78.95,6.00),v60,z5,tPen\WObj:=wPaper;
    MoveL Offs(pOrigin,230.88,78.50,6.00),vTravel,z5,tPen\WObj:=wPaper;
  ENDPROC

  PROC DrawPart152()
    MoveL Offs(pOrigin,230.88,78.50,0.00),v60,z0,tPen\WObj:=wPaper;
    MoveL Offs(pOrigin,227.88,81.51,0.00),v40,z0,tPen\WObj:=wPaper;
    MoveL Offs(pOrigin,228.35,80.80,0.00),v40,z0,tPen\WObj:=wPaper;
    MoveL Offs(pOrigin,231.36,83.80,0.00),v40,z0,tPen\WObj:=wPaper;
    MoveL Offs(pOrigin,230.88,83.64,0.00),v40,z0,tPen\WObj:=wPaper;
    MoveL Offs(pOrigin,229.18,83.64,0.00),v40,z0,tPen\WObj:=wPaper;
    MoveL Offs(pOrigin,229.39,84.70,0.00),v40,z0,tPen\WObj:=wPaper;
    MoveL Offs(pOrigin,230.66,84.70,0.00),v40,z0,tPen\WObj:=wPaper;
    MoveL Offs(pOrigin,230.22,84.69,0.00),v40,z0,tPen\WObj:=wPaper;
    MoveL Offs(pOrigin,230.22,82.35,0.00),v40,z0,tPen\WObj:=wPaper;
    MoveL Offs(pOrigin,230.88,82.14,0.00),v40,z0,tPen\WObj:=wPaper;
    MoveL Offs(pOrigin,230.88,85.54,0.00),v40,z0,tPen\WObj:=wPaper;
    MoveL Offs(pOrigin,231.73,91.28,0.00),v40,z0,tPen\WObj:=wPaper;
    MoveL Offs(pOrigin,232.79,103.81,0.00),v40,z0,tPen\WObj:=wPaper;
    MoveL Offs(pOrigin,233.00,118.26,0.00),v40,z0,tPen\WObj:=wPaper;
    MoveL Offs(pOrigin,231.94,136.96,0.00),v40,z0,tPen\WObj:=wPaper;
    MoveL Offs(pOrigin,228.96,164.80,0.00),v40,z0,tPen\WObj:=wPaper;
    MoveL Offs(pOrigin,229.81,164.95,0.00),v40,z0,tPen\WObj:=wPaper;
    MoveL Offs(pOrigin,227.48,164.95,0.00),v40,z0,tPen\WObj:=wPaper;
    MoveL Offs(pOrigin,226.96,164.53,0.00),v40,z0,tPen\WObj:=wPaper;
    MoveL Offs(pOrigin,229.82,167.39,0.00),v40,z0,tPen\WObj:=wPaper;
    MoveL Offs(pOrigin,229.39,167.14,0.00),v40,z0,tPen\WObj:=wPaper;
    MoveL Offs(pOrigin,228.75,166.71,0.00),v40,z0,tPen\WObj:=wPaper;
    MoveL Offs(pOrigin,228.96,165.23,0.00),v40,z0,tPen\WObj:=wPaper;
    MoveL Offs(pOrigin,230.24,163.95,0.00),v40,z0,tPen\WObj:=wPaper;
    MoveL Offs(pOrigin,230.24,163.95,0.00),v40,z0,tPen\WObj:=wPaper;
    MoveL Offs(pOrigin,230.24,163.10,0.00),v40,z0,tPen\WObj:=wPaper;
    MoveL Offs(pOrigin,231.09,162.68,0.00),v40,z0,tPen\WObj:=wPaper;
    MoveL Offs(pOrigin,231.09,162.68,0.00),v40,z0,tPen\WObj:=wPaper;
    MoveL Offs(pOrigin,231.30,161.40,0.00),v40,z0,tPen\WObj:=wPaper;
    MoveL Offs(pOrigin,230.84,160.95,0.00),v40,z0,tPen\WObj:=wPaper;
    MoveL Offs(pOrigin,231.90,162.00,0.00),v40,z0,tPen\WObj:=wPaper;
    MoveL Offs(pOrigin,232.28,162.23,0.00),v40,z0,tPen\WObj:=wPaper;
    MoveL Offs(pOrigin,225.81,168.70,0.00),v40,fine,tPen\WObj:=wPaper;
    MoveL Offs(pOrigin,225.81,168.70,6.00),v60,z5,tPen\WObj:=wPaper;
    MoveL Offs(pOrigin,226.38,169.92,6.00),vTravel,z5,tPen\WObj:=wPaper;
    MoveL Offs(pOrigin,226.38,169.92,0.00),v60,z0,tPen\WObj:=wPaper;
    MoveL Offs(pOrigin,229.38,172.93,0.00),v40,z0,tPen\WObj:=wPaper;
    MoveL Offs(pOrigin,229.55,172.43,0.00),v40,z0,tPen\WObj:=wPaper;
    MoveL Offs(pOrigin,224.89,177.09,0.00),v40,z0,tPen\WObj:=wPaper;
    MoveL Offs(pOrigin,225.50,176.51,0.00),v40,z0,tPen\WObj:=wPaper;
    MoveL Offs(pOrigin,230.31,181.32,0.00),v40,z0,tPen\WObj:=wPaper;
    MoveL Offs(pOrigin,230.72,181.71,0.00),v40,z0,tPen\WObj:=wPaper;
    MoveL Offs(pOrigin,227.86,184.57,0.00),v40,z0,tPen\WObj:=wPaper;
    MoveL Offs(pOrigin,228.22,183.71,0.00),v40,z0,tPen\WObj:=wPaper;
    MoveL Offs(pOrigin,233.03,188.52,0.00),v40,z0,tPen\WObj:=wPaper;
    MoveL Offs(pOrigin,232.19,189.20,0.00),v40,z0,tPen\WObj:=wPaper;
    MoveL Offs(pOrigin,244.36,177.03,0.00),v40,z0,tPen\WObj:=wPaper;
    MoveL Offs(pOrigin,243.93,177.02,0.00),v40,z0,tPen\WObj:=wPaper;
    MoveL Offs(pOrigin,242.27,175.36,0.00),v40,z0,tPen\WObj:=wPaper;
    MoveL Offs(pOrigin,241.82,175.09,0.00),v40,z0,tPen\WObj:=wPaper;
    MoveL Offs(pOrigin,254.60,162.32,0.00),v40,z0,tPen\WObj:=wPaper;
    MoveL Offs(pOrigin,255.34,163.06,0.00),v40,z0,tPen\WObj:=wPaper;
    MoveL Offs(pOrigin,250.83,167.57,0.00),v40,z0,tPen\WObj:=wPaper;
    MoveL Offs(pOrigin,250.49,167.15,0.00),v40,z0,tPen\WObj:=wPaper;
    MoveL Offs(pOrigin,249.14,165.80,0.00),v40,z0,tPen\WObj:=wPaper;
    MoveL Offs(pOrigin,249.58,166.01,0.00),v40,z0,tPen\WObj:=wPaper;
    MoveL Offs(pOrigin,250.85,166.01,0.00),v40,z0,tPen\WObj:=wPaper;
    MoveL Offs(pOrigin,251.23,166.40,0.00),v40,z0,tPen\WObj:=wPaper;
    MoveL Offs(pOrigin,249.88,165.05,0.00),v40,z0,tPen\WObj:=wPaper;
    MoveL Offs(pOrigin,249.50,164.43,0.00),v40,z0,tPen\WObj:=wPaper;
    MoveL Offs(pOrigin,243.33,170.59,0.00),v40,z0,tPen\WObj:=wPaper;
    MoveL Offs(pOrigin,243.76,170.87,0.00),v40,z0,tPen\WObj:=wPaper;
    MoveL Offs(pOrigin,245.26,172.38,0.00),v40,z0,tPen\WObj:=wPaper;
    MoveL Offs(pOrigin,245.88,172.53,0.00),v40,z0,tPen\WObj:=wPaper;
    MoveL Offs(pOrigin,235.51,182.90,0.00),v40,z0,tPen\WObj:=wPaper;
    MoveL Offs(pOrigin,234.76,182.15,0.00),v40,z0,tPen\WObj:=wPaper;
    MoveL Offs(pOrigin,239.72,177.19,0.00),v40,z0,tPen\WObj:=wPaper;
    MoveL Offs(pOrigin,239.12,176.29,0.00),v40,z0,tPen\WObj:=wPaper;
    MoveL Offs(pOrigin,234.31,181.10,0.00),v40,fine,tPen\WObj:=wPaper;
    MoveL Offs(pOrigin,234.31,181.10,6.00),v60,z5,tPen\WObj:=wPaper;
    MoveL Offs(pOrigin,234.17,179.75,6.00),vTravel,z5,tPen\WObj:=wPaper;
    MoveL Offs(pOrigin,234.17,179.75,0.00),v60,z0,tPen\WObj:=wPaper;
    MoveL Offs(pOrigin,238.23,175.70,0.00),v40,z0,tPen\WObj:=wPaper;
    MoveL Offs(pOrigin,237.25,175.21,0.00),v40,z0,tPen\WObj:=wPaper;
    MoveL Offs(pOrigin,232.15,178.54,0.00),v40,z0,tPen\WObj:=wPaper;
    MoveL Offs(pOrigin,231.30,178.82,0.00),v40,z0,tPen\WObj:=wPaper;
    MoveL Offs(pOrigin,230.95,178.61,0.00),v40,z0,tPen\WObj:=wPaper;
    MoveL Offs(pOrigin,231.16,177.55,0.00),v40,z0,tPen\WObj:=wPaper;
    MoveL Offs(pOrigin,234.91,173.30,0.00),v40,z0,tPen\WObj:=wPaper;
    MoveL Offs(pOrigin,235.90,172.80,0.00),v40,z0,tPen\WObj:=wPaper;
    MoveL Offs(pOrigin,240.86,167.35,0.00),v40,fine,tPen\WObj:=wPaper;
    MoveL Offs(pOrigin,240.86,167.35,6.00),v60,z5,tPen\WObj:=wPaper;
    MoveL Offs(pOrigin,239.15,167.31,6.00),vTravel,z5,tPen\WObj:=wPaper;
    MoveL Offs(pOrigin,239.15,167.31,0.00),v60,z0,tPen\WObj:=wPaper;
    MoveL Offs(pOrigin,244.26,162.20,0.00),v40,fine,tPen\WObj:=wPaper;
    MoveL Offs(pOrigin,244.26,162.20,6.00),v60,z5,tPen\WObj:=wPaper;
    MoveL Offs(pOrigin,245.15,164.29,6.00),vTravel,z5,tPen\WObj:=wPaper;
    MoveL Offs(pOrigin,245.15,164.29,0.00),v60,z0,tPen\WObj:=wPaper;
    MoveL Offs(pOrigin,223.21,186.23,0.00),v40,z0,tPen\WObj:=wPaper;
    MoveL Offs(pOrigin,223.43,186.39,0.00),v40,z0,tPen\WObj:=wPaper;
    MoveL Offs(pOrigin,225.39,188.34,0.00),v40,z0,tPen\WObj:=wPaper;
    MoveL Offs(pOrigin,224.92,188.18,0.00),v40,z0,tPen\WObj:=wPaper;
    MoveL Offs(pOrigin,223.65,188.18,0.00),v40,z0,tPen\WObj:=wPaper;
    MoveL Offs(pOrigin,223.29,187.74,0.00),v40,z0,tPen\WObj:=wPaper;
    MoveL Offs(pOrigin,225.09,189.54,0.00),v40,z0,tPen\WObj:=wPaper;
    MoveL Offs(pOrigin,224.71,189.24,0.00),v40,z0,tPen\WObj:=wPaper;
    MoveL Offs(pOrigin,223.44,189.24,0.00),v40,z0,tPen\WObj:=wPaper;
    MoveL Offs(pOrigin,223.14,189.09,0.00),v40,z0,tPen\WObj:=wPaper;
    MoveL Offs(pOrigin,224.79,190.74,0.00),v40,z0,tPen\WObj:=wPaper;
    MoveL Offs(pOrigin,224.50,190.30,0.00),v40,z0,tPen\WObj:=wPaper;
    MoveL Offs(pOrigin,223.22,190.30,0.00),v40,z0,tPen\WObj:=wPaper;
    MoveL Offs(pOrigin,222.70,190.13,0.00),v40,z0,tPen\WObj:=wPaper;
    MoveL Offs(pOrigin,224.65,192.09,0.00),v40,z0,tPen\WObj:=wPaper;
    MoveL Offs(pOrigin,224.08,192.41,0.00),v40,z0,tPen\WObj:=wPaper;
    MoveL Offs(pOrigin,222.80,192.41,0.00),v40,z0,tPen\WObj:=wPaper;
    MoveL Offs(pOrigin,222.25,192.68,0.00),v40,z0,tPen\WObj:=wPaper;
    MoveL Offs(pOrigin,224.06,194.48,0.00),v40,z0,tPen\WObj:=wPaper;
    MoveL Offs(pOrigin,223.44,194.52,0.00),v40,z0,tPen\WObj:=wPaper;
    MoveL Offs(pOrigin,222.16,194.52,0.00),v40,z0,tPen\WObj:=wPaper;
    MoveL Offs(pOrigin,221.81,193.73,0.00),v40,z0,tPen\WObj:=wPaper;
    MoveL Offs(pOrigin,223.76,195.68,0.00),v40,z0,tPen\WObj:=wPaper;
    MoveL Offs(pOrigin,223.44,195.58,0.00),v40,z0,tPen\WObj:=wPaper;
    MoveL Offs(pOrigin,221.52,195.58,0.00),v40,z0,tPen\WObj:=wPaper;
    MoveL Offs(pOrigin,221.52,195.40,0.00),v40,z0,tPen\WObj:=wPaper;
    MoveL Offs(pOrigin,222.09,194.98,0.00),v40,z0,tPen\WObj:=wPaper;
    MoveL Offs(pOrigin,222.59,193.49,0.00),v40,z0,tPen\WObj:=wPaper;
    MoveL Offs(pOrigin,225.35,180.10,0.00),v40,z0,tPen\WObj:=wPaper;
    MoveL Offs(pOrigin,228.75,154.39,0.00),v40,z0,tPen\WObj:=wPaper;
    MoveL Offs(pOrigin,231.09,128.89,0.00),v40,z0,tPen\WObj:=wPaper;
  ENDPROC

  PROC DrawPart153()
    MoveL Offs(pOrigin,231.51,119.32,0.00),v40,z0,tPen\WObj:=wPaper;
    MoveL Offs(pOrigin,231.51,108.70,0.00),v40,z0,tPen\WObj:=wPaper;
    MoveL Offs(pOrigin,230.66,95.31,0.00),v40,z0,tPen\WObj:=wPaper;
    MoveL Offs(pOrigin,229.60,86.39,0.00),v40,z0,tPen\WObj:=wPaper;
    MoveL Offs(pOrigin,227.90,75.97,0.00),v40,z0,tPen\WObj:=wPaper;
    MoveL Offs(pOrigin,225.77,66.20,0.00),v40,z0,tPen\WObj:=wPaper;
    MoveL Offs(pOrigin,223.65,58.34,0.00),v40,z0,tPen\WObj:=wPaper;
    MoveL Offs(pOrigin,221.45,51.75,0.00),v40,z0,tPen\WObj:=wPaper;
    MoveL Offs(pOrigin,220.89,51.25,0.00),v40,z0,tPen\WObj:=wPaper;
    MoveL Offs(pOrigin,217.98,54.09,0.00),v40,z0,tPen\WObj:=wPaper;
    MoveL Offs(pOrigin,218.12,57.28,0.00),v40,z0,tPen\WObj:=wPaper;
    MoveL Offs(pOrigin,217.27,59.61,0.00),v40,z0,tPen\WObj:=wPaper;
    MoveL Offs(pOrigin,218.12,68.96,0.00),v40,z0,tPen\WObj:=wPaper;
    MoveL Offs(pOrigin,218.12,80.65,0.00),v40,z0,tPen\WObj:=wPaper;
    MoveL Offs(pOrigin,217.27,90.43,0.00),v40,z0,tPen\WObj:=wPaper;
    MoveL Offs(pOrigin,215.57,101.05,0.00),v40,z0,tPen\WObj:=wPaper;
    MoveL Offs(pOrigin,212.81,112.53,0.00),v40,z0,tPen\WObj:=wPaper;
    MoveL Offs(pOrigin,202.82,147.80,0.00),v40,z0,tPen\WObj:=wPaper;
    MoveL Offs(pOrigin,195.18,176.91,0.00),v40,z0,tPen\WObj:=wPaper;
    MoveL Offs(pOrigin,196.24,177.83,0.00),v40,z0,tPen\WObj:=wPaper;
    MoveL Offs(pOrigin,209.62,184.92,0.00),v40,z0,tPen\WObj:=wPaper;
    MoveL Offs(pOrigin,212.60,186.97,0.00),v40,z0,tPen\WObj:=wPaper;
    MoveL Offs(pOrigin,213.02,187.68,0.00),v40,z0,tPen\WObj:=wPaper;
    MoveL Offs(pOrigin,213.59,187.82,0.00),v40,z0,tPen\WObj:=wPaper;
    MoveL Offs(pOrigin,213.88,188.81,0.00),v40,z0,tPen\WObj:=wPaper;
    MoveL Offs(pOrigin,213.88,188.81,0.00),v40,z0,tPen\WObj:=wPaper;
    MoveL Offs(pOrigin,221.31,195.40,0.00),v40,z0,tPen\WObj:=wPaper;
    MoveL Offs(pOrigin,221.74,196.25,0.00),v40,z0,tPen\WObj:=wPaper;
    MoveL Offs(pOrigin,220.25,204.11,0.00),v40,z0,tPen\WObj:=wPaper;
    MoveL Offs(pOrigin,219.61,210.49,0.00),v40,z0,tPen\WObj:=wPaper;
    MoveL Offs(pOrigin,218.76,211.98,0.00),v40,z0,tPen\WObj:=wPaper;
    MoveL Offs(pOrigin,218.34,212.19,0.00),v40,z0,tPen\WObj:=wPaper;
    MoveL Offs(pOrigin,217.91,212.33,0.00),v40,z0,tPen\WObj:=wPaper;
    MoveL Offs(pOrigin,217.27,211.98,0.00),v40,z0,tPen\WObj:=wPaper;
    MoveL Offs(pOrigin,213.02,207.51,0.00),v40,z0,tPen\WObj:=wPaper;
    MoveL Offs(pOrigin,198.29,190.09,0.00),v40,z0,tPen\WObj:=wPaper;
    MoveL Offs(pOrigin,198.57,189.52,0.00),v40,z0,tPen\WObj:=wPaper;
    MoveL Offs(pOrigin,208.56,186.05,0.00),v40,z0,tPen\WObj:=wPaper;
    MoveL Offs(pOrigin,209.62,186.19,0.00),v40,z0,tPen\WObj:=wPaper;
    MoveL Offs(pOrigin,212.60,188.18,0.00),v40,z0,tPen\WObj:=wPaper;
    MoveL Offs(pOrigin,212.60,188.18,0.00),v40,z0,tPen\WObj:=wPaper;
    MoveL Offs(pOrigin,213.88,188.81,0.00),v40,fine,tPen\WObj:=wPaper;
    MoveL Offs(pOrigin,213.88,188.81,6.00),v60,z5,tPen\WObj:=wPaper;
    MoveL Offs(pOrigin,212.72,189.26,6.00),vTravel,z5,tPen\WObj:=wPaper;
    MoveL Offs(pOrigin,212.72,189.26,0.00),v60,z0,tPen\WObj:=wPaper;
    MoveL Offs(pOrigin,214.52,187.45,0.00),v40,z0,tPen\WObj:=wPaper;
    MoveL Offs(pOrigin,213.62,186.86,0.00),v40,z0,tPen\WObj:=wPaper;
    MoveL Offs(pOrigin,211.67,188.81,0.00),v40,z0,tPen\WObj:=wPaper;
    MoveL Offs(pOrigin,212.36,188.75,0.00),v40,z0,tPen\WObj:=wPaper;
    MoveL Offs(pOrigin,206.49,182.89,0.00),v40,z0,tPen\WObj:=wPaper;
    MoveL Offs(pOrigin,206.01,182.90,0.00),v40,z0,tPen\WObj:=wPaper;
    MoveL Offs(pOrigin,203.68,182.90,0.00),v40,z0,tPen\WObj:=wPaper;
    MoveL Offs(pOrigin,203.68,183.29,0.00),v40,z0,tPen\WObj:=wPaper;
    MoveL Offs(pOrigin,204.10,183.50,0.00),v40,z0,tPen\WObj:=wPaper;
    MoveL Offs(pOrigin,203.68,183.29,0.00),v40,z0,tPen\WObj:=wPaper;
    MoveL Offs(pOrigin,203.15,183.89,0.00),v40,z0,tPen\WObj:=wPaper;
    MoveL Offs(pOrigin,205.40,181.64,0.00),v40,z0,tPen\WObj:=wPaper;
    MoveL Offs(pOrigin,204.52,182.23,0.00),v40,z0,tPen\WObj:=wPaper;
    MoveL Offs(pOrigin,204.95,182.44,0.00),v40,z0,tPen\WObj:=wPaper;
    MoveL Offs(pOrigin,204.52,182.23,0.00),v40,z0,tPen\WObj:=wPaper;
    MoveL Offs(pOrigin,203.89,181.85,0.00),v40,z0,tPen\WObj:=wPaper;
    MoveL Offs(pOrigin,201.76,181.85,0.00),v40,z0,tPen\WObj:=wPaper;
    MoveL Offs(pOrigin,202.19,182.44,0.00),v40,z0,tPen\WObj:=wPaper;
    MoveL Offs(pOrigin,202.82,182.86,0.00),v40,z0,tPen\WObj:=wPaper;
    MoveL Offs(pOrigin,202.19,182.44,0.00),v40,z0,tPen\WObj:=wPaper;
    MoveL Offs(pOrigin,201.85,182.73,0.00),v40,z0,tPen\WObj:=wPaper;
    MoveL Offs(pOrigin,196.89,177.77,0.00),v40,z0,tPen\WObj:=wPaper;
    MoveL Offs(pOrigin,196.66,178.19,0.00),v40,z0,tPen\WObj:=wPaper;
    MoveL Offs(pOrigin,197.09,178.40,0.00),v40,z0,tPen\WObj:=wPaper;
    MoveL Offs(pOrigin,196.66,178.19,0.00),v40,z0,tPen\WObj:=wPaper;
    MoveL Offs(pOrigin,195.81,177.76,0.00),v40,z0,tPen\WObj:=wPaper;
    MoveL Offs(pOrigin,196.24,177.98,0.00),v40,z0,tPen\WObj:=wPaper;
    MoveL Offs(pOrigin,195.81,177.76,0.00),v40,z0,tPen\WObj:=wPaper;
    MoveL Offs(pOrigin,195.81,177.62,0.00),v40,z0,tPen\WObj:=wPaper;
    MoveL Offs(pOrigin,194.32,177.62,0.00),v40,z0,tPen\WObj:=wPaper;
    MoveL Offs(pOrigin,194.11,178.19,0.00),v40,z0,tPen\WObj:=wPaper;
    MoveL Offs(pOrigin,194.54,178.40,0.00),v40,z0,tPen\WObj:=wPaper;
    MoveL Offs(pOrigin,194.11,178.19,0.00),v40,z0,tPen\WObj:=wPaper;
    MoveL Offs(pOrigin,193.58,178.53,0.00),v40,z0,tPen\WObj:=wPaper;
    MoveL Offs(pOrigin,196.43,175.68,0.00),v40,z0,tPen\WObj:=wPaper;
    MoveL Offs(pOrigin,195.99,175.37,0.00),v40,z0,tPen\WObj:=wPaper;
    MoveL Offs(pOrigin,194.18,173.57,0.00),v40,z0,tPen\WObj:=wPaper;
    MoveL Offs(pOrigin,193.59,174.04,0.00),v40,z0,tPen\WObj:=wPaper;
    MoveL Offs(pOrigin,197.95,169.68,0.00),v40,z0,tPen\WObj:=wPaper;
    MoveL Offs(pOrigin,197.47,169.38,0.00),v40,z0,tPen\WObj:=wPaper;
    MoveL Offs(pOrigin,195.66,167.58,0.00),v40,z0,tPen\WObj:=wPaper;
    MoveL Offs(pOrigin,195.11,168.04,0.00),v40,z0,tPen\WObj:=wPaper;
    MoveL Offs(pOrigin,199.62,163.53,0.00),v40,z0,tPen\WObj:=wPaper;
    MoveL Offs(pOrigin,198.95,163.40,0.00),v40,z0,tPen\WObj:=wPaper;
    MoveL Offs(pOrigin,197.29,161.74,0.00),v40,z0,tPen\WObj:=wPaper;
    MoveL Offs(pOrigin,197.94,161.78,0.00),v40,z0,tPen\WObj:=wPaper;
    MoveL Offs(pOrigin,199.00,161.78,0.00),v40,z0,tPen\WObj:=wPaper;
    MoveL Offs(pOrigin,199.39,162.35,0.00),v40,z0,tPen\WObj:=wPaper;
    MoveL Offs(pOrigin,197.59,160.55,0.00),v40,z0,tPen\WObj:=wPaper;
    MoveL Offs(pOrigin,198.15,160.73,0.00),v40,z0,tPen\WObj:=wPaper;
    MoveL Offs(pOrigin,199.21,160.73,0.00),v40,z0,tPen\WObj:=wPaper;
    MoveL Offs(pOrigin,199.54,161.00,0.00),v40,z0,tPen\WObj:=wPaper;
    MoveL Offs(pOrigin,197.88,159.35,0.00),v40,z0,tPen\WObj:=wPaper;
    MoveL Offs(pOrigin,198.36,159.67,0.00),v40,z0,tPen\WObj:=wPaper;
    MoveL Offs(pOrigin,199.42,159.67,0.00),v40,z0,tPen\WObj:=wPaper;
    MoveL Offs(pOrigin,199.98,159.95,0.00),v40,z0,tPen\WObj:=wPaper;
    MoveL Offs(pOrigin,198.18,158.15,0.00),v40,z0,tPen\WObj:=wPaper;
    MoveL Offs(pOrigin,197.68,158.00,0.00),v40,z0,tPen\WObj:=wPaper;
    MoveL Offs(pOrigin,202.19,153.49,0.00),v40,z0,tPen\WObj:=wPaper;
    MoveL Offs(pOrigin,201.91,152.92,0.00),v40,z0,tPen\WObj:=wPaper;
    MoveL Offs(pOrigin,199.96,150.97,0.00),v40,z0,tPen\WObj:=wPaper;
    MoveL Offs(pOrigin,200.49,151.22,0.00),v40,z0,tPen\WObj:=wPaper;
    MoveL Offs(pOrigin,201.76,151.22,0.00),v40,z0,tPen\WObj:=wPaper;
    MoveL Offs(pOrigin,202.20,151.72,0.00),v40,z0,tPen\WObj:=wPaper;
    MoveL Offs(pOrigin,200.40,149.92,0.00),v40,z0,tPen\WObj:=wPaper;
    MoveL Offs(pOrigin,200.91,150.17,0.00),v40,z0,tPen\WObj:=wPaper;
    MoveL Offs(pOrigin,201.98,150.17,0.00),v40,z0,tPen\WObj:=wPaper;
    MoveL Offs(pOrigin,202.35,150.37,0.00),v40,z0,tPen\WObj:=wPaper;
    MoveL Offs(pOrigin,200.70,148.72,0.00),v40,z0,tPen\WObj:=wPaper;
    MoveL Offs(pOrigin,201.12,149.11,0.00),v40,z0,tPen\WObj:=wPaper;
    MoveL Offs(pOrigin,202.19,149.11,0.00),v40,z0,tPen\WObj:=wPaper;
    MoveL Offs(pOrigin,202.80,149.33,0.00),v40,z0,tPen\WObj:=wPaper;
    MoveL Offs(pOrigin,201.14,147.67,0.00),v40,z0,tPen\WObj:=wPaper;
    MoveL Offs(pOrigin,201.34,148.06,0.00),v40,z0,tPen\WObj:=wPaper;
    MoveL Offs(pOrigin,202.61,148.06,0.00),v40,z0,tPen\WObj:=wPaper;
  ENDPROC

